    // Application specific
    xIN_PickPiece : BOOL; (* signal from the pick and place element
                             the number of picked signal depend on the recipe *)
    xIN_RotTableBlockedByPnp : BOOL; // Is the pick and place blocking the rotary table?
END_VAR
VAR_OUTPUT
    (* standart Ausgänge *)
    xOUT_ErrFlag  : BOOL;           // Error Flag 
    xOUT_Busy     : BOOL;           // Baustein befindet sich im Ablauf 
    xOUT_Done     : BOOL;           // Baustein hat den Ablauf beendet 		
    xOUT_Ready    : BOOL;           // Ready to begin, should be the same state as done	
    xOUT_Timeout  : BOOL;           // Timeout FB 
    xOUT_InitDone : BOOL;           // initialisierung fertig
    xOUT_Wait     : BOOL;           // Wartet auf Bedingung
    iOUT_Step     : ST125_Feeder_e; // Aktueller Schritt 
    sOUT_Step     : STRING;         // Aktueller Schritt but in string format
    bOUT_Error    : BYTE;           // Fehlernummer

    // Application specific
    xOUT_PceReadyToPick : BOOL; // the piece(s) is/are ready to picked
END_VAR
VAR
    (* Standard *)
    (* Schritt *)
    iLastStep : ST125_Feeder_e; // Merker letzter Schritt 
    iPreStep  : ST125_Feeder_e; // Schritt zurück nach Alarm 
    iAktStep  : ST125_Feeder_e; // aktueller Schritt

    // Trigger Starten 
    rtSTART : R_TRIG;
    // Timer TimeOut 
    TON_Timeout : TON;

    (* Bausteine *)

    // Application specific
    fb_axis125_10W               : FB_AxisLMturn_V1_1;
    simu_axis125_10W             : FB_Simu_AxisLM_V1_1;
    fb_feeder                    : FB_Feeder2Sensors;
    fifo                         : FB_Fifo(3);
    simu_feeder                  : FB_Simu_Feeder; // simulation of a feeder
    simu_fifo_feeder_to_rotTable : FB_Fifo(30);    // fifo to hold a piece
    rtPutPiece                   : R_TRIG;         // trigger to add a piece

    rtPick : R_TRIG; // r_trig signal from the pick and place machine

    iCurrentTableIndex : INT; // current table index
    iSearchIndex       : INT; (* Initialization index TO see how many element we have AT startup
                                 or after an alarm *)

    xPieceInSeparator      : BOOL; // The piece is at the entry of the round table
    xPieceWrongInSeparator : BOOL; // A piece is detected at the separator but it is the wrong one

    // This ton is used to ensure that the piece is completely inside
    // the entry of the round table so we are sure that we mesure correctly the piece up to
    // the top
    TON_waitForControl : TON;

END_VAR
VAR CONSTANT
    MAX_SEARCH_TURN : INT := 3; // maximum search number

    FEEDER_SIMULATION : BOOL := FALSE; // Simulate this code
END_VAR

(*******************************************************************)
(* Trigger  *)
(*******************************************************************)
(* Zurücksetzen *)
IF xIN_RESET THEN
    iPreStep  := ST125_Feeder_e.RESET;
    iOUT_Step := ST125_Feeder_e.RESET;
END_IF;

(* Error Quittieren *)
IF (bOUT_Error <> 0) AND xIN_Quit THEN
    xOUT_ErrFlag := FALSE;
    bOUT_Error   := 0;
    iOUT_Step    := iPreStep;
END_IF;

iCurrentTableIndex := iCurrentTableIndex MOD 3;

(*******************************************************************)
(* Timer *)
(*******************************************************************)
TON_Timeout(IN := xIN_NextStep AND (iLastStep = iOUT_Step) (*todo FG *) ,
            PT := tIN_Timeout);

xPieceInSeparator := (IN.AI21_ST125_piece_height < _20_AUTO.recipe.st125.diPieceGoodMaxHeight) AND
                     (IN.AI21_ST125_piece_height > _20_AUTO.recipe.st125.diPieceGoodMinHeight);

xPieceWrongInSeparator := (IN.AI21_ST125_piece_height < _20_AUTO.recipe.st125.diPieceWrongMaxHeight) AND
                          (IN.AI21_ST125_piece_height > _20_AUTO.recipe.st125.diPieceWrongMinHeight);

TON_waitForControl(IN := xPieceInSeparator,
                   PT := DINT_TO_TIME(_20_AUTO.recipe.st125.TON_WaitPieceTime));

(*******************************************************************)
(* Bausteine *)
(*******************************************************************)

fb_feeder(xIN_Enable                := enIN_State = enState.StateAUTO OR enIN_State = enState.StateSTEP,
          xIN_PieceInEnd            := IO_BOX.I8401_ST125_maximum_wf,
          xIN_PieceMax              := IO_BOX.I8401_ST125_maximum_wf,
          xIN_InSimulation          := FEEDER_SIMULATION AND CONST.USE_SIMULATION,
          refIN_SimulatedFifo       := simu_fifo_feeder_to_rotTable,
          iIN_FifoSetMaxSensorValue := 20,
          diIN_SignlFilter_ms       := _20_AUTO.recipe.st125.FeederConfig.InFilterDelay,
          diIN_StartDelay_ms        := _20_AUTO.recipe.st125.FeederConfig.StartDelay,
          diIN_StopDelay_ms         := _20_AUTO.recipe.st125.FeederConfig.StopDelay,
          diIN_EmptyDelay_ms        := _20_AUTO.recipe.st125.FeederConfig.EmptyDelay);

simu_feeder(xIN_Enable         := fb_feeder.xOUT_EnableFeeder AND FEEDER_SIMULATION AND CONST.USE_SIMULATION,
            xIN_PceSensor      := fb_feeder.xIN_PieceMax,
            tIN_NewPieceTime   := 500,
            iIN_WaitTimeMin_ms := 500,
            iIN_WaitTimeMax_ms := 1000);

rtPick(CLK := xIN_PickPiece);
rtPutPiece(CLK := simu_feeder.xOUT_NewPiece);

IF rtPutPiece.Q AND NOT simu_fifo_feeder_to_rotTable.IsFull() THEN
    simu_fifo_feeder_to_rotTable.Put(1);
END_IF

IF ST125_Feeder_e.Init_simu_home_table = iOUT_Step THEN
    fb_axis125_10W.rIN_Position := TO_REAL(120.0 - LMOD(ST125_Axis.axis125_10W.rActPos, 120.0));

ELSE
    fb_axis125_10W.rIN_Position := 120.0;

END_IF

simu_axis125_10W(xIN_Enable          := FEEDER_SIMULATION AND CONST.USE_SIMULATION,
                 wIN_AxisState       := ST125_Axis.axis125_10W.wState,
                 bIN_AxisCntr        := fb_axis125_10W.bOUT_AxisCntr,
                 udiIN_HomingTime_ms := 1000,
                 pIN_axisSimu        := ADR(SIMU.axis_ref[Axis_e.ST125_10W]),
                 pIN_axisHW          := ADR(ST125_Axis.axis125_10W.axis),
                 rIN_PosActual       := fb_axis125_10W.rOUT_ActPos,
                 rIN_PosMax          := ST125_Axis.const125_10W.POS_MAX,
                 rIN_PosMin          := ST125_Axis.const125_10W.POS_MIN,
                 rIN_PixMax          := 0,
                 rIN_PixMin          := 0);

fb_axis125_10W(enIN_State     := enIN_State,
               parIN_Buttons  := ADR(AXIS.btTeachArAxis[Axis_e.ST125_10W]),
               xIN_DisButtons :=,
               xIN_Quit       := xIN_Quit,
               xIN_PARAMok    := TRUE,
               xIN_FREE       := NOT xIN_RotTableBlockedByPnp,
               xIN_FREE_HOME  := TRUE,
               rIN_POSMIN     := ST125_Axis.const125_10W.POS_MIN,
               rIN_POSMAX     := ST125_Axis.const125_10W.POS_MAX,
               rIN_VELOMAX    := ST125_Axis.const125_10W.VELO_MAX,
               rIN_VELOMANU   := ST125_Axis.const125_10W.VELO_MANU,
               rIN_VELOOPEN   := ST125_Axis.const125_10W.VELO_MANU / 4,
               rIN_JogInc     := AXIS.rTeachIncAxis,
               xIN_Execute    := ST125_Feeder_e.Init_set_table_pos = iOUT_Step OR
                                 ST125_Feeder_e.Init_table_go_to_zero = iOUT_Step OR
                                 ST125_Feeder_e.Init_simu_home_table = iOUT_Step OR
                                 ST125_Feeder_e.load_piece = iOUT_Step OR
                                 ST125_Feeder_e.wait_rotary_table_done = iOUT_Step,
               xIN_Relative     := fb_axis125_10W.xIN_Execute,
               xIN_STOP         := FALSE,
               xIN_OFF          := FALSE,
               rIN_Position     :=, // Is set above
               rIN_Velocity     := TO_REAL(100.0),
               rIN_Acceleration := TO_REAL(2160.0),
               rIN_Deceleration := TO_REAL(2160.0),
               rIN_Jerk         := TO_REAL(720000.0),
               xIN_Home         := ST125_feeder_e.Init_home_table = iOUT_Step,
               xIN_Reset        := xIN_Reset OR ST125_feeder_e.RESET = iOUT_Step,
               // The simu fb gives us the hardware signal when we are not in simulation
               wAxisState    := simu_axis125_10W.wOUT_AxisState,
               bOUT_AxisCntr => ST125_Axis.axis125_10W.bCtrlHi,
               rOUT_ActPos   =>, // leave empty, rActPos must be set using the modulo
               axisIN_REF    := simu_axis125_10W.pOUT_axisRef^);

ST125_Axis.axis125_10W.rActPos := LREAL_TO_REAL(simu_axis125_10W.pOUT_axisRef^.NcToPlc.ModuloActPos);

(*******************************************************************)
(* OUTPUTS *)
(*******************************************************************)
// Error Flag 
xOUT_ErrFlag := (bOUT_Error <> 0) OR (ST125_Feeder_e.ERROR = iOUT_Step);
// Baustein befindet sich im Ablauf 
xOUT_Busy := (iOUT_Step > ST125_Feeder_e.READY) AND (iOUT_Step < ST125_Feeder_e.DONE);
// Baustein hat den Ablauf beendet
xOUT_Done := (iOUT_Step = ST125_Feeder_e.DONE);
// Process ready
xOUT_Ready := (iOUT_Step = ST125_Feeder_e.READY);
// Timeout FB 				 		
xOUT_Timeout := TON_Timeout.Q;
// Itialisierung fertig			
xOUT_InitDone := (iOUT_Step = ST125_Feeder_e.READY);
// Aktueller Schritt			
iOUT_Step := iOUT_Step; //Im Ablauf gesetzt		
sOUT_Step := TO_STRING(iOUT_Step);
//Fehlernummer	 
bOUT_Error := bOUT_Error; //Im Ablauf/FB gesetzt	
(* Warte (alle Schritte wo auf FG oder Teile gewartet wird) *)
xOUT_Wait := (iOUT_Step = ST125_Feeder_e.DONE) OR
             (iOUT_Step = ST125_Feeder_e.READY);

IO_BOX.Q8402_ST125_freigabe_wf := fb_feeder.xOUT_EnableFeeder AND NOT (FEEDER_SIMULATION AND CONST.USE_SIMULATION);

IO_BOX.Q8400_ST125_freigabe_REO :=
    (IO_BOX.Q8402_ST125_freigabe_wf OR
    (ST125_Feeder_e.wait_on_a_piece = iOUT_Step) OR
    (ST125_Feeder_e.DONE = iOUT_Step AND NOT xPieceInSeparator)) AND
    NOT (FEEDER_SIMULATION AND CONST.USE_SIMULATION);

(*******************************************************************)
(* Ablauf *)
(*******************************************************************)

(* Sperren *)
IF xIN_Sperre THEN
    iPreStep  := ST125_Feeder_e.RESET;
    iOUT_Step := ST125_Feeder_e.RESET;
    RETURN;
END_IF;

(* Schritt Merker *)
IF iAktStep <> iOUT_Step THEN
    iLastStep := iAktStep;
    iAktStep  := iOUT_Step;
END_IF

(* START *)
rtSTART(CLK := xIN_Start);

IF 0 = bOUT_Error THEN
    IF fb_axis125_10W.xOUT_ErrFlag THEN 
        bOUT_Error := ST125_Alarm_e.Axis_120_10W_error;
        iPreStep   := ST145_Feeder_e.INIT;
		
    ELSIF fb_feeder.xOUT_Empty THEN
        bOUT_Error := ST125_Alarm_e.Feeder_empty;
        iPreStep   := ST145_Feeder_e.READY;
		
	ELSIF IN.I504_distanzsensor_verschmutzung_125 THEN
        bOUT_Error := ST125_Alarm_e.Distance_sensor_dirty;
        iPreStep   := ST145_Feeder_e.INIT;
	
    END_IF
ELSIF iOUT_Step < ST125_Feeder_e.ERROR THEN
    iOUT_Step := ST125_Feeder_e.ERROR;
END_IF

(*******************************************************************)
(* Schrittkette  *)
(*******************************************************************)
CASE iOUT_Step OF

(***** RESET *****)
ST125_Feeder_e.RESET: (* Schritt 0-99 *)
    //Initialisierungen
    //Start Init Ablauf
    IF xIN_Init THEN
        iOUT_Step := ST125_Feeder_e.INIT;
        //Start Manu Ablauf
    ELSIF enIN_State = StateMANU AND xIN_NextStep THEN
        iOUT_Step := ST125_Feeder_e.INIT;
    END_IF;

(***** INIT *****)
ST125_Feeder_e.INIT: (* Grundstellung ? *)
    IF NOT xIN_RotTableBlockedByPnp THEN
        iOUT_Step := ST125_Feeder_e.Init_home_table;
    END_IF

ST125_Feeder_e.Init_home_table:
    IF fb_axis125_10W.xOUT_HOMED THEN
        iCurrentTableIndex := 0;

        IF FEEDER_SIMULATION AND CONST.USE_SIMULATION THEN
            iOUT_Step := ST125_Feeder_e.Init_simu_home_table;
        ELSE
            iOUT_Step := ST125_Feeder_e.Init_reset_search_index;
        END_IF
    END_IF

ST125_Feeder_e.Init_simu_home_table:
    IF fb_axis125_10W.xOUT_DONE THEN
        iOUT_Step := ST125_Feeder_e.Init_reset_search_index;
    END_IF

// unused, done by the drive itself, see drive configuration
ST125_Feeder_e.Init_table_go_to_zero:
    IF fb_axis125_10W.xOUT_DONE THEN
        iOUT_Step := ST125_Feeder_e.Init_reset_search_index;
    END_IF

ST125_Feeder_e.Init_reset_search_index:
    iSearchIndex := 0;
    fifo.Empty();
    iOUT_Step := ST125_Feeder_e.READY; // Bypass search algorithm, unusful

ST125_Feeder_e.Init_set_table_pos:
    IF fb_axis125_10W.xOUT_DONE THEN
        iCurrentTableIndex := iCurrentTableIndex + 1;
        iOUT_Step          := ST125_Feeder_e.Init_see_if_piece_there;
    END_IF

ST125_Feeder_e.Init_see_if_piece_there:
    IF simu_feeder.xOUT_NewPiece THEN
        fifo.Put(1);
    END_IF

    IF iSearchIndex < MAX_SEARCH_TURN THEN
        iOUT_Step    := ST125_Feeder_e.Init_set_table_pos;
        iSearchIndex := iSearchIndex + 1;
    ELSE
        iOUT_Step := ST125_Feeder_e.READY;
    END_IF

(***** READY / INIT DONE *****)
ST125_Feeder_e.READY: (* Start AUTO,END,LEER,STEP *)
    IF xIN_Start THEN //IF rtSTART.Q THEN
        iOUT_Step := ST125_Feeder_e.START;
    END_IF

(***** START  ZYKLISCH *****)
ST125_Feeder_e.START: (*  *)
    IF xIN_NextStep AND pxFG_Freigabe^ THEN
        iOUT_Step := ST125_Feeder_e.check_if_feeding_necessary;
    END_IF;

ST125_Feeder_e.check_if_feeding_necessary:
    IF fifo.IsFull() THEN
        iOUT_Step := ST125_Feeder_e.DONE;
    ELSE
        iOUT_Step := ST125_Feeder_e.wait_on_a_piece;
    END_IF

ST125_Feeder_e.wait_on_a_piece:
    IF (FEEDER_SIMULATION AND CONST.USE_SIMULATION AND NOT simu_fifo_feeder_to_rotTable.IsEmpty()) OR
       (NOT (FEEDER_SIMULATION AND CONST.USE_SIMULATION) AND TON_waitForControl.Q) THEN
        iOUT_Step := ST125_Feeder_e.load_piece;
        simu_fifo_feeder_to_rotTable.Pop(1);
    END_IF

ST125_Feeder_e.load_piece:
    IF NOT fb_axis125_10W.xOUT_DONE THEN
        iOUT_Step := ST125_Feeder_e.wait_rotary_table_done;
    END_IF

ST125_Feeder_e.wait_rotary_table_done:
    IF fb_axis125_10W.xOUT_DONE THEN
        fifo.Put(1);
        iOUT_Step := ST125_Feeder_e.check_if_feeding_necessary;
    END_IF

(***** DONE *****)
ST125_Feeder_e.DONE: (* Letzter Schritt  *)
    IF rtPick.Q THEN
        fifo.Pop(TO_INT(_20_AUTO.recipe.st125.xUseVerLeft));
        fifo.Pop(TO_INT(_20_AUTO.recipe.st125.xUseVerRight));
    END_IF

    IF NOT xIN_AlarmAktiv THEN
        //AUTO
        IF (enIN_State = StateAUTO) AND xIN_RestartCYCL AND NOT fifo.IsFull() THEN
            iOUT_Step := ST125_Feeder_e.START;
            //STEP / END / LEERFAHREN restart
        ELSIF (enIN_State < StateAUTO) AND (enIN_State >= enState.StateSTEP) AND xIN_RestartCYCL AND NOT fifo.IsFull()
            THEN
            iOUT_Step := ST125_Feeder_e.START;
            //STEP / END / LEERFAHREN fertig
        ELSIF (enIN_State = StateREADY) THEN
            iOUT_Step := ST125_Feeder_e.READY;
        END_IF;
    END_IF;

(************ ERROR *************)
ST125_Feeder_e.ERROR: (* ERROR *) ;

END_CASE;

END_FUNCTION_BLOCK

// ---- POUs/20_AUTO/ST125/POU_ALARM_125.TcPOU
PROGRAM POU_ALARM_125
VAR_INPUT
    xIN_QUIT      : BOOL; // Alarm quittieren
    iIN_ArraySize : INT;
    pstrIN_ALARM  : POINTER TO structAlarm;       // Array Alarmstruktur
    refPOU        : REFERENCE TO FB_AUT_ABSTRACT; // the POU to test
END_VAR
VAR_OUTPUT
    xOUT_AL_ST : BOOL; // Alarm Station aktiv
END_VAR
VAR
    //Alarmbaustein
    _FB_ALARM_ST : FB_ALARM;
    //Local
    iIndex : INT; // Index For Schleife	
END_VAR
VAR CONSTANT
    sDefString : STRING := 'Error ST120,'; // Station #
END_VAR

(********************** INITIALISIERE VARIABLEN ****************************)
FOR iIndex := 0 TO iIN_ArraySize - 1 DO
    pstrIN_ALARM[iIndex].xAlarmIN   := FALSE;
    pstrIN_ALARM[iIndex].xAlarmOFF  := FALSE;
    pstrIN_ALARM[iIndex].xAlarmSAVE := TRUE;
    pstrIN_ALARM[iIndex].xAlarmQUIT := xIN_QUIT;
    pstrIN_ALARM[iIndex].tAlarmVERZ := T#100MS;
    pstrIN_ALARM[iIndex].sAlarmText := '';
    pstrIN_ALARM[iIndex].bAlarmNr   := 0;
END_FOR

(********************** ALARME ****************************)
pstrIN_ALARM[0].xAlarmIN   := (refPOU.bOUT_ErrorNum = ST120_Alarm_e.Axis_120_01Y_error);
pstrIN_ALARM[0].sAlarmText := CONCAT(sDefString, ' Axis 01Y in error');
pstrIN_ALARM[0].bAlarmNr   := 0;

pstrIN_ALARM[1].xAlarmIN   := (refPOU.bOUT_ErrorNum = ST120_Alarm_e.Axis_120_02Z_error);
pstrIN_ALARM[1].sAlarmText := CONCAT(sDefString, ' Axis 02Z in error');
pstrIN_ALARM[1].bAlarmNr   := 0;

pstrIN_ALARM[2].xAlarmIN   := (refPOU.bOUT_ErrorNum = ST120_Alarm_e.Cylinder_griper_left);
pstrIN_ALARM[2].sAlarmText := CONCAT(sDefString, ' Cylinder .05 gripper right');
pstrIN_ALARM[2].bAlarmNr   := 0;

pstrIN_ALARM[3].xAlarmIN   := (refPOU.bOUT_ErrorNum = ST120_Alarm_e.Cylinder_griper_right);
pstrIN_ALARM[3].sAlarmText := CONCAT(sDefString, ' Cylinder .06 gripper left');
pstrIN_ALARM[3].bAlarmNr   := 0;

pstrIN_ALARM[7].xAlarmIN   := (refPOU.bOUT_ErrorNum = ST120_Alarm_e.Feeder_error);
pstrIN_ALARM[7].sAlarmText := CONCAT(sDefString, ' One part of the feeder is in error');
pstrIN_ALARM[7].bAlarmNr   := 0;

pstrIN_ALARM[8].xAlarmIN   := (refPOU.bOUT_ErrorNum = ST120_Alarm_e.Piece_in_unused_griper);
pstrIN_ALARM[8].sAlarmText := CONCAT(sDefString, ' One part is handled by a unused griper');
pstrIN_ALARM[8].bAlarmNr   := 0;

pstrIN_ALARM[9].xAlarmIN   := (refPOU.bOUT_ErrorNum = ST120_Alarm_e.Piece_missing_left_griper);
pstrIN_ALARM[9].sAlarmText := CONCAT(sDefString, ' A piece is missing in the left griper');
pstrIN_ALARM[9].bAlarmNr   := 0;

pstrIN_ALARM[10].xAlarmIN   := (refPOU.bOUT_ErrorNum = ST120_Alarm_e.Piece_missing_right_griper);
pstrIN_ALARM[10].sAlarmText := CONCAT(sDefString, ' A piece is missing in the right griper');
pstrIN_ALARM[10].bAlarmNr   := 0;

pstrIN_ALARM[11].xAlarmIN   := (refPOU.bOUT_ErrorNum = ST120_Alarm_e.Feeder_empty);
pstrIN_ALARM[11].sAlarmText := CONCAT(sDefString, ' The feeder is empty');
pstrIN_ALARM[11].bAlarmNr   := 0;

(********************** ALARM FB ****************************)
_FB_ALARM_ST(pstrIN_Alarm  := pstrIN_ALARM,
             iIN_ArraySize := ST120_Alarm_e._max);

(********************** ALARM FB ****************************)
xOUT_AL_ST := FALSE;

FOR iIndex := 0 TO iIN_ArraySize - 1 DO
    IF pstrIN_ALARM[iIndex].xAlarmOUT THEN
        xOUT_AL_ST := TRUE;
    END_IF
END_FOR

END_PROGRAM

// ---- POUs/20_AUTO/ST128/FB_AUT_128.TcPOU
FUNCTION_BLOCK FB_AUT_128 EXTENDS FB_AUT_ABSTRACT
(****************************************************************************)
(*	POU_AUT_zxx			Bausteinaufrufe Station	zxx							*)
(*	Status				ungetestet											*)
(*  Version:			1.0													*)
(*	Beschrieb:																*)
(*																			*)
(*	Abläufe:			FB_ABLzxxA		Hauptablauf							*)
(*																			*)
(*																			*)
(* 	25.09.2019/Dj															*)
(****************************************************************************)
(*	dd.mm.yyyy   KZ    x.y			Beschrieb								*)
(****************************************************************************)
VAR_INPUT
    (* spezifische Eingänge *)

END_VAR
VAR_OUTPUT
    (* spezifische Ausgänge *)

END_VAR
VAR
    (* Bausteine *)
    fb_TubeCapCheck : FB_ABL_128_TubeCapCheck; // 
END_VAR

(*******************************************************************)
(* Timer *)
(*******************************************************************)

(*******************************************************************)
(* Flanken / Merker *)
(*******************************************************************)
//MANU CYCLE
IF (enIN_State = StateMANU) AND xIN_ManuCycle THEN
    xManuCycle := TRUE;
END_IF;

IF (enIN_State <> StateMANU) OR xOUT_Done THEN
    xManuCycle := FALSE;
END_IF

//NEXT STEP
xNextStep := (enIN_State > StateSTEP) OR
             ((enIN_State = StateSTEP) AND xIN_Step) OR
             ((enIN_State = StateMANU) AND xManuCycle);

//RESET
xReset := (enIN_State < StateREADY) AND (enIN_State <> StateINIT) AND NOT xManuCycle;

(*******************************************************************)
(* Bausteinaufrufe Abläufe *)
(*******************************************************************)

xRelease := MAIN.MoverMan.IsProcessUsed(THIS^);

fb_TubeCapCheck(xIN_Reset       := xReset,
                xIN_Init        := xIN_Init,
                xIN_Quit        := xIN_Quit,
                xIN_Start       := enIN_State >= enState.StateLEER AND xRelease,
                xIN_Sperre      := NOT xIN_On,
                xIN_NextStep    := xNextStep,
                xIN_AlarmAktiv  := xIN_AlarmAktiv,
                xIN_DryCycle    := xIN_DryCycle,
                xIN_RestartCYCL := enIN_State >= enState.StateLEER,
                enIN_State      := enIN_State,
                tIN_Timeout     := tIN_Timeout,
                pxFG_Freigabe   := ADR(xRelease),
                Mover           := THIS^.Mover);

(*******************************************************************)
(* Mover reset flags *)
(*******************************************************************)

(*******************************************************************)
(* OUTPUT *)
(*******************************************************************)
xOUT_InitDone := fb_TubeCapCheck.xOUT_InitDone;
xOUT_Ready    := fb_TubeCapCheck.xOUT_Ready;
xOUT_Done     := fb_TubeCapCheck.xOUT_Done;
xOUT_ErrFlag  := fb_TubeCapCheck.xOUT_ErrFlag;
xOUT_Wait     := fb_TubeCapCheck.xOUT_Wait;
xOUT_AlarmST  := xOUT_ErrFlag;

(*******************************************************************)
(* Bausteinaufruf Error Station *)
(*******************************************************************)
// POU_ERR_VORLAGE(xIN_QUIT:=xIN_Quit , pstrArIN_ALARM:=ADR(HMI.strArALARM[1]));

(* % of completion of the process *)
PROPERTY iCompletionPC : INT
GET
iCompletionPC := THIS^.fb_TubeCapCheck.iOUT_ProcessCompletion;
END_GET
END_PROPERTY

PROPERTY ProcessExecution : ProcessExecution_e
GET
ProcessExecution := THIS^._ProcessExecution;
END_GET
SET
THIS^._ProcessExecution := ProcessExecution;
END_SET
END_PROPERTY

PROPERTY xBusy : BOOL
GET
xBusy := THIS^.fb_TubeCapCheck.xOUT_Busy;
END_GET
SET
END_SET
END_PROPERTY

PROPERTY xDone : BOOL
GET
xDone := THIS^.fb_TubeCapCheck.xOUT_Ready OR THIS^.fb_TubeCapCheck.xOUT_Done;
END_GET
END_PROPERTY

PROPERTY xMoverPathFree : BOOL
GET
xMoverPathFree := THIS^.fb_TubeCapCheck.xOUT_MoverFree OR THIS^.fb_TubeCapCheck.xOUT_Ready OR THIS^.fb_TubeCapCheck.xOUT_Done;
END_GET
END_PROPERTY

PROPERTY xMoverShouldLeave : BOOL
GET
xMoverShouldLeave := THIS^.fb_TubeCapCheck.iOUT_Step = ST128_TubeCapCheck_e.SYNC_MOVER_LEAVE;
END_GET
END_PROPERTY

END_FUNCTION_BLOCK

// ---- POUs/20_AUTO/ST128/FB_ABL_128_TubeCapCheck.TcPOU
FUNCTION_BLOCK FB_ABL_128_TubeCapCheck
(****************************************************************************************)
(*	TITEL				laden kristall- Modul	    										*)
(*	Status				ungetestet                         								*)
(*	Beschrieb:			Ablaufbeschreibung												*)
(*																						*)
(*	Steps:	self-explained using enum													*)
(***********************************Revisionen*******************************************)
(*	see github blames																	*)
(****************************************************************************************)

VAR_INPUT
    xIN_Reset       : BOOL;          // Schrittkette zurücksetzen 
    xIN_Init        : BOOL;          // Initialisieren
    xIN_Quit        : BOOL;          // Fehler quittieren 
    xIN_Start       : BOOL;          // Startbefehl
    xIN_Sperre      : BOOL;          // FB Sperren 
    xIN_NextStep    : BOOL;          // Nächsten Schritt ausführen 
    xIN_AlarmAktiv  : BOOL;          // Anlage hat Alarm
    xIN_DryCycle    : BOOL;          // Fahren ohne Teile
    xIN_RestartCYCL : BOOL;          // Zyklus erneut starten im STEP: END: LEERFAHREN
    enIN_State      : enState;       // Status Anlage
    tIN_Timeout     : TIME := T#10s; // Timout

    pxFG_Freigabe : POINTER TO BOOL; //Freigabe von Station

    // Application specific
    Mover : REFERENCE TO FB_Mover;
END_VAR
VAR_OUTPUT
    (* standart Ausgänge *)
    xOUT_ErrFlag  : BOOL;                 // Error Flag 
    xOUT_Busy     : BOOL;                 // Baustein befindet sich im Ablauf 
    xOUT_Done     : BOOL;                 // Baustein hat den Ablauf beendet 		
    xOUT_Ready    : BOOL;                 // Ready to begin: should be the same state as done	
    xOUT_Timeout  : BOOL;                 // Timeout FB 
    xOUT_InitDone : BOOL;                 // initialisierung fertig
    xOUT_Wait     : BOOL;                 // Wartet auf Bedingung
    iOUT_Step     : ST128_TubeCapCheck_e; // Aktueller Schritt 
    sOUT_Step     : STRING;               // Aktueller Schritt but in string format
    bOUT_Error    : BYTE;                 // Fehlernummer

    iOUT_ProcessCompletion : INT;  //process completion: express in % (0-100)
    xOUT_MoverFree         : BOOL; // The mover is free to move

END_VAR
VAR
    (* Standard *)
    (* Schritt *)
    iLastStep : ST128_TubeCapCheck_e; // Merker letzter Schritt 
    iPreStep  : ST128_TubeCapCheck_e; // Schritt zurück nach Alarm 
    iAktStep  : ST128_TubeCapCheck_e; // aktueller Schritt

    // Trigger Starten 
    rtSTART : R_TRIG;
    // Timer TimeOut 
    TON_Timeout : TON;

    (* Bausteine *)
    ton_WaitInPosMin : TON;  // protect the inpos flag to come to early
    capFoundRight    : BOOL; // TRUE when all measured level are OK
    capFoundLeft     : BOOL; // TRUE when all measured level are OK

    visu_shuttle_x_position : LREAL; // position of the shuttle used in visu

END_VAR
VAR CONSTANT
    TUBE_CAP_CHECK_SIMULATION : BOOL := FALSE; // Set to TRUE to simulate this part of the program
END_VAR

(*******************************************************************)
(* Trigger  *)
(*******************************************************************)
(* Zurücksetzen *)
IF xIN_RESET THEN
    iPreStep  := ST128_TubeCapCheck_e.RESET;
    iOUT_Step := ST128_TubeCapCheck_e.RESET;
END_IF;

(* Error Quittieren *)
IF (bOUT_Error <> 0) AND xIN_Quit THEN
    xOUT_ErrFlag := FALSE;
    bOUT_Error   := 0;
    iOUT_Step    := iPreStep; // iPreStep;
END_IF;

(*******************************************************************)
(* Timer *)
(*******************************************************************)
TON_Timeout(IN := xIN_NextStep AND (iLastStep = iOUT_Step) (*todo FG *) ,
            PT := tIN_Timeout);

ton_WaitInPosMin(IN := __ISVALIDREF(Mover) AND_THEN Mover.IsInStationPos(), PT := T#100MS);

(*******************************************************************)
(* Bausteine *)
(*******************************************************************)
IF (iOUT_Step = ST128_TubeCapCheck_e.Wait_move_and_check_tube_cap_right OR
   iOUT_Step = ST128_TubeCapCheck_e.Move_shuttle_relative_right) AND
   IO_BOX.I2000_ST128_filterhut_vorhanden THEN
    capFoundRight := TRUE;
END_IF

IF (iOUT_Step = ST128_TubeCapCheck_e.Wait_move_and_check_tube_cap_left OR
   iOUT_Step = ST128_TubeCapCheck_e.Move_shuttle_relative_left) AND
   IO_BOX.I2000_ST128_filterhut_vorhanden THEN
    capFoundLeft := TRUE;
END_IF

(*******************************************************************)
(* OUTPUTS *)
(*******************************************************************)
// Error Flag 
xOUT_ErrFlag := (bOUT_Error <> 0) OR (ST128_TubeCapCheck_e.ERROR = iOUT_Step);
// Baustein befindet sich im Ablauf 
xOUT_Busy := (iOUT_Step > ST128_TubeCapCheck_e.READY) AND (iOUT_Step < ST128_TubeCapCheck_e.DONE);
// Baustein hat den Ablauf beendet
xOUT_Done := (iOUT_Step = ST128_TubeCapCheck_e.DONE);
// Process ready
xOUT_Ready := (iOUT_Step = ST128_TubeCapCheck_e.READY);
// Timeout FB 				 		
xOUT_Timeout := TON_Timeout.Q;
// Itialisierung fertig			
xOUT_InitDone := (iOUT_Step = ST128_TubeCapCheck_e.READY) OR
                 (iOUT_Step = ST128_TubeCapCheck_e.DONE);

// Aktueller Schritt			
iOUT_Step := iOUT_Step; //Im Ablauf gesetzt		
sOUT_Step := TO_STRING(iOUT_Step);
//Fehlernummer	 
bOUT_Error := bOUT_Error; //Im Ablauf/FB gesetzt	
(* Warte (alle Schritte wo auf FG oder Teile gewartet wird) *)
xOUT_Wait := (iOUT_Step = ST128_TubeCapCheck_e.DONE) OR
             (iOUT_Step = ST128_TubeCapCheck_e.READY) OR
             (iOUT_Step = ST128_TubeCapCheck_e.START) OR
             (iOUT_Step = ST128_TubeCapCheck_e.waitOnMover) OR
             (iOUT_Step = ST128_TubeCapCheck_e.SYNC_MOVER_LEAVE);

xOUT_MoverFree :=
    NOT ((iOUT_Step >= ST128_TubeCapCheck_e.MOVER_NEEDED_OP) AND (iOUT_Step < ST128_TubeCapCheck_e.MOVER_FREE_OP)) AND
    (iOUT_Step >= ST128_TubeCapCheck_e.READY) AND
    (iOUT_Step < ST128_TubeCapCheck_e.ERROR);

iOUT_ProcessCompletion := F_GetPercent_2(iOUT_Step,
                                         ST128_TubeCapCheck_e.waitOnMover,
                                         ST128_TubeCapCheck_e.DONE,
                                         ST128_TubeCapCheck_e.waitOnMover,
                                         ST128_TubeCapCheck_e.DONE);

(*******************************************************************)
(* Ablauf *)
(*******************************************************************)

(* Sperren *)
IF xIN_Sperre THEN
    iPreStep  := ST128_TubeCapCheck_e.RESET;
    iOUT_Step := ST128_TubeCapCheck_e.RESET;
    RETURN;
END_IF;

(* Schritt Merker *)
IF iAktStep <> iOUT_Step THEN
    iLastStep := iAktStep;
    iAktStep  := iOUT_Step;
END_IF

(* START *)
rtSTART(CLK := xIN_Start);

IF __ISVALIDREF(Mover) THEN
    visu_shuttle_x_position := Mover.MovingProcessOffset;
ELSE
    visu_shuttle_x_position := 0.0;
END_IF

IF 0 = bOUT_Error THEN
    // put error conditions here
ELSIF iOUT_Step < ST128_TubeCapCheck_e.ERROR THEN
    iOUT_Step := ST128_TubeCapCheck_e.ERROR;
END_IF

(*******************************************************************)
(* Schrittkette  *)
(*******************************************************************)
CASE iOUT_Step OF

(***** RESET *****)
ST128_TubeCapCheck_e.RESET: (* Schritt 0-99 *)
    //Initialisierungen
    //Start Init Ablauf
    IF xIN_Init THEN
        iOUT_Step := ST128_TubeCapCheck_e.INIT;
        //Start Manu Ablauf
    ELSIF enIN_State = StateMANU AND xIN_NextStep THEN
        iOUT_Step := ST128_TubeCapCheck_e.INIT;
    END_IF;

(***** INIT *****)
ST128_TubeCapCheck_e.INIT: (* Grundstellung ? *)
    iOUT_Step := ST128_TubeCapCheck_e.READY;

(***** READY / INIT DONE *****)
ST128_TubeCapCheck_e.READY: (* Start AUTO:END:LEER:STEP *)
    IF xIN_Start THEN       //IF rtSTART.Q THEN
        iOUT_Step := ST128_TubeCapCheck_e.START;
    END_IF

(***** START  ZYKLISCH *****)
ST128_TubeCapCheck_e.START: (*  *)
    IF xIN_NextStep AND pxFG_Freigabe^ THEN
        iOUT_Step     := ST128_TubeCapCheck_e.waitOnMover;
        capFoundRight := FALSE;
        capFoundLeft  := FALSE;
    END_IF;

ST128_TubeCapCheck_e.waitOnMover:
    IF xIN_NextStep AND __ISVALIDREF(Mover) OR HMI.bArForceCyclusState[StationList_e.ST128] THEN
        IF Mover.GetLastStationDone() >= INT#128 THEN
            iOUT_Step := ST128_TubeCapCheck_e.SYNC_MOVER_LEAVE;
        ELSIF Mover.GetLastStationDone() < INT#125 THEN
            iOUT_Step := ST128_TubeCapCheck_e.SYNC_MOVER_LEAVE;
        ELSE
            iOUT_Step := ST128_TubeCapCheck_e.Move_shuttle_relative_right;
        END_IF
    END_IF

ST128_TubeCapCheck_e.Move_shuttle_relative_right:
    IF __ISVALIDREF(Mover) THEN
        IF Mover.MoveRelativeInsideStation(40.0) THEN
            iOUT_Step := ST128_TubeCapCheck_e.Wait_move_and_check_tube_cap_right;
            iPreStep  := ST128_TubeCapCheck_e.Wait_move_and_check_tube_cap_right;
        END_IF
    ELSE
        bOUT_Error := 10;
    END_IF

ST128_TubeCapCheck_e.Wait_move_and_check_tube_cap_right:
    IF xIN_NextStep AND __ISVALIDREF(Mover) AND_THEN ton_WaitInPosMin.Q THEN
        IF _20_AUTO.recipe.st128.xIsTypeMiniOrSmart THEN
            iOUT_Step := ST128_TubeCapCheck_e.Move_shuttle_to_pos_left;
        ELSE
            iOUT_Step := ST128_TubeCapCheck_e.Save_result_in_mover;
            iPreStep  := ST128_TubeCapCheck_e.Save_result_in_mover;
        END_IF
    END_IF

ST128_TubeCapCheck_e.Move_shuttle_to_pos_left:
    IF __ISVALIDREF(Mover) THEN
        IF Mover.MoveRelativeInsideStation(60.0) THEN
            iOUT_Step := ST128_TubeCapCheck_e.Wait_move_done_pos_left;
            iPreStep  := ST128_TubeCapCheck_e.Wait_move_done_pos_left;
        END_IF
    ELSE
        bOUT_Error := 11;
    END_IF

ST128_TubeCapCheck_e.Wait_move_done_pos_left:
    IF xIN_NextStep AND __ISVALIDREF(Mover) AND_THEN ton_WaitInPosMin.Q THEN
        iOUT_Step := ST128_TubeCapCheck_e.Move_shuttle_relative_left;
    END_IF

ST128_TubeCapCheck_e.Move_shuttle_relative_left:
    IF __ISVALIDREF(Mover) THEN
        IF Mover.MoveRelativeInsideStation(40.0) THEN
            iOUT_Step := ST128_TubeCapCheck_e.Wait_move_and_check_tube_cap_left;
            iPreStep  := ST128_TubeCapCheck_e.Wait_move_and_check_tube_cap_left;
        END_IF
    ELSE
        bOUT_Error := 12;
    END_IF

ST128_TubeCapCheck_e.Wait_move_and_check_tube_cap_left:
    IF xIN_NextStep AND __ISVALIDREF(Mover) AND_THEN ton_WaitInPosMin.Q THEN
        iOUT_Step := ST128_TubeCapCheck_e.Save_result_in_mover;
    END_IF

ST128_TubeCapCheck_e.Save_result_in_mover:
    IF (NOT capFoundRight OR
       (_20_AUTO.recipe.st128.xIsTypeMiniOrSmart AND NOT capFoundLeft)) AND
       NOT (TUBE_CAP_CHECK_SIMULATION AND CONST.USE_SIMULATION) THEN
        iOUT_Step := ST128_TubeCapCheck_e.ERROR;

        IF __ISVALIDREF(Mover) THEN

            IF NOT capFoundLeft AND NOT capFoundRight THEN
                Mover.SetErrorCode('128-B Left and Right');

            ELSIF capFoundLeft THEN
                Mover.SetErrorCode('128-B Left');

            ELSIF capFoundRight THEN
                Mover.SetErrorCode('128-B Right');

            ELSE
                ASSERT(0); // Read your code again, you should never go here !

            END_IF

            IF NOT Mover.SetLastStation(-128) THEN
                ASSERT(0);
            END_IF
        END_IF

        bOUT_Error := 1;
        iPreStep   := ST128_TubeCapCheck_e.SYNC_MOVER_LEAVE;
    ELSE
        iOUT_Step := ST128_TubeCapCheck_e.SYNC_MOVER_LEAVE;

        IF __ISVALIDREF(Mover) THEN
            IF NOT Mover.SetLastStation(128) THEN
                ASSERT(0);
            END_IF
        END_IF
    END_IF

ST128_TubeCapCheck_e.SYNC_MOVER_LEAVE:
    // The mover needs to be taken by MoverMan
    IF NOT __ISVALIDREF(Mover) THEN
        iOUT_Step := ST128_TubeCapCheck_e.DONE;
    END_IF

(***** DONE *****)
ST128_TubeCapCheck_e.DONE: (* Letzter Schritt  *)
    IF NOT xIN_AlarmAktiv THEN
        //AUTO
        IF (enIN_State = StateAUTO) AND xIN_RestartCYCL THEN
            iOUT_Step := ST128_TubeCapCheck_e.START;
            //STEP / END / LEERFAHREN restart
        ELSIF (enIN_State < StateAUTO) AND (enIN_State >= enState.StateSTEP) AND xIN_RestartCYCL THEN
            iOUT_Step := ST128_TubeCapCheck_e.START;
            //STEP / END / LEERFAHREN fertig
        ELSIF (enIN_State = StateREADY) THEN
            iOUT_Step := ST128_TubeCapCheck_e.READY;
        END_IF;
    END_IF;

(************ ERROR *************)
ST128_TubeCapCheck_e.ERROR: (* ERROR *) ;

END_CASE;

END_FUNCTION_BLOCK

// ---- POUs/20_AUTO/ST130/FB_AUT_130.TcPOU
FUNCTION_BLOCK FB_AUT_130 EXTENDS FB_AUT_ABSTRACT
(****************************************************************************)
(*	POU_AUT_zxx			Bausteinaufrufe Station	zxx							*)
(*	Status				ungetestet											*)
(*  Version:			1.0													*)
(*	Beschrieb:																*)
(*																			*)
(*	Abläufe:			FB_ABLzxxA		Hauptablauf							*)
(*																			*)
(*																			*)
(* 	25.09.2019/Dj															*)
(****************************************************************************)
(*	dd.mm.yyyy   KZ    x.y			Beschrieb								*)
(****************************************************************************)
VAR_INPUT
    (* spezifische Eingänge *)

END_VAR
VAR_OUTPUT
    (* spezifische Ausgänge *)

END_VAR
VAR
    (* Bausteine *)
    fb_Dose : FB_ABL_130_Dose;

    fb_stat : FB_AUT_Statistics;

END_VAR

(*******************************************************************)
(* Timer *)
(*******************************************************************)

(*******************************************************************)
(* Flanken / Merker *)
(*******************************************************************)
//MANU CYCLE
IF (enIN_State = StateMANU) AND xIN_ManuCycle THEN
    xManuCycle := TRUE;
END_IF;

IF (enIN_State <> StateMANU) OR xOUT_Done THEN
    xManuCycle := FALSE;
END_IF

//NEXT STEP
xNextStep := (enIN_State > StateSTEP) OR
             ((enIN_State = StateSTEP) AND xIN_Step) OR
             ((enIN_State = StateMANU) AND xManuCycle);

//RESET
xReset := (enIN_State < StateREADY) AND (enIN_State <> StateINIT) AND NOT xManuCycle;

(*******************************************************************)
(* Bausteinaufrufe Abläufe *)
(*******************************************************************)

xRelease := MAIN.MoverMan.IsProcessUsed(THIS^);

fb_Dose(xIN_Reset       := xReset,
        xIN_Init        := xIN_Init,
        xIN_Quit        := xIN_Quit,
        xIN_Start       := enIN_State >= enState.StateLEER AND xRelease,
        xIN_Sperre      := NOT xIN_On,
        xIN_NextStep    := xNextStep,
        xIN_AlarmAktiv  := xIN_AlarmAktiv,
        xIN_DryCycle    := xIN_DryCycle,
        xIN_RestartCYCL := enIN_State >= enState.StateLEER,
        enIN_State      := enIN_State,
        tIN_Timeout     := tIN_Timeout,
        pxFG_Freigabe   := ADR(xRelease),
        Mover           := THIS^.Mover);

fb_stat(xIN_Enable  := enState.StateAUTO = enIN_State,
        xIN_Waiting := fb_Dose.xOUT_Wait,
        xIN_Running := (fb_Dose.iOUT_Step >= ST130_Dose_e.START) AND
                       (fb_Dose.iOUT_Step <= ST130_Dose_e.DONE),
        // Since we use a mover system, a cycle is done when we are waiting on a mover
        xIN_Done := fb_Dose.iOUT_Step = ST130_Dose_e.waitOnMover);

(*******************************************************************)
(* Mover reset flags *)
(*******************************************************************)

(*******************************************************************)
(* OUTPUT *)
(*******************************************************************)
xOUT_InitDone := fb_Dose.xOUT_InitDone;
xOUT_Ready    := fb_Dose.xOUT_Ready;
xOUT_Done     := fb_Dose.xOUT_Done;
xOUT_ErrFlag  := fb_Dose.xOUT_ErrFlag;
xOUT_Wait     := fb_Dose.xOUT_Wait;
xOUT_AlarmST  := xOUT_ErrFlag;

(*******************************************************************)
(* Bausteinaufruf Error Station *)
(*******************************************************************)
// POU_ERR_VORLAGE(xIN_QUIT:=xIN_Quit , pstrArIN_ALARM:=ADR(HMI.strArALARM[1]));

(* % of completion of the process *)
PROPERTY iCompletionPC : INT
GET
iCompletionPC := THIS^.fb_Dose.iOUT_ProcessCompletion;
END_GET
END_PROPERTY

PROPERTY ProcessExecution : ProcessExecution_e
GET
ProcessExecution := THIS^._ProcessExecution;
END_GET
SET
THIS^._ProcessExecution := ProcessExecution;
END_SET
END_PROPERTY

PROPERTY xBusy : BOOL
GET
xBusy := THIS^.fb_Dose.xOUT_Busy;
END_GET
SET
END_SET
END_PROPERTY

PROPERTY xDone : BOOL
GET
xDone := THIS^.fb_Dose.xOUT_Ready OR THIS^.fb_Dose.xOUT_Done;
END_GET
END_PROPERTY

PROPERTY xMoverPathFree : BOOL
GET
xMoverPathFree := THIS^.fb_Dose.xOUT_MoverFree OR THIS^.fb_Dose.xOUT_Ready OR THIS^.fb_Dose.xOUT_Done;
END_GET
END_PROPERTY

PROPERTY xMoverShouldLeave : BOOL
GET
xMoverShouldLeave := THIS^.fb_Dose.iOUT_Step = ST130_Dose_e.SYNC_MOVER_LEAVE;
END_GET
END_PROPERTY

END_FUNCTION_BLOCK

// ---- POUs/20_AUTO/ST130/FB_ABL_130_Dose.TcPOU
FUNCTION_BLOCK FB_ABL_130_Dose
(****************************************************************************************)
(*	TITEL				laden kristall- Modul	    										*)
(*	Status				ungetestet                         								*)
(*	Beschrieb:			Ablaufbeschreibung												*)
(*																						*)
(*	Steps:	self-explained using enum													*)
(***********************************Revisionen*******************************************)
(*	see github blames																	*)
(****************************************************************************************)

VAR_INPUT
    xIN_Reset       : BOOL;          // Schrittkette zurücksetzen 
    xIN_Init        : BOOL;          // Initialisieren
    xIN_Quit        : BOOL;          // Fehler quittieren 
    xIN_Start       : BOOL;          // Startbefehl
    xIN_Sperre      : BOOL;          // FB Sperren 
    xIN_NextStep    : BOOL;          // Nächsten Schritt ausführen 
    xIN_AlarmAktiv  : BOOL;          // Anlage hat Alarm
    xIN_DryCycle    : BOOL;          // Fahren ohne Teile
    xIN_RestartCYCL : BOOL;          // Zyklus erneut starten im STEP: END: LEERFAHREN
    enIN_State      : enState;       // Status Anlage
    tIN_Timeout     : TIME := T#10s; // Timout

    pxFG_Freigabe : POINTER TO BOOL; //Freigabe von Station

    // Application specific
    Mover : REFERENCE TO FB_Mover;
END_VAR
VAR_OUTPUT
    (* standart Ausgänge *)
    xOUT_ErrFlag  : BOOL;         // Error Flag 
    xOUT_Busy     : BOOL;         // Baustein befindet sich im Ablauf 
    xOUT_Done     : BOOL;         // Baustein hat den Ablauf beendet 		
    xOUT_Ready    : BOOL;         // Ready to begin: should be the same state as done	
    xOUT_Timeout  : BOOL;         // Timeout FB 
    xOUT_InitDone : BOOL;         // initialisierung fertig
    xOUT_Wait     : BOOL;         // Wartet auf Bedingung
    iOUT_Step     : ST130_Dose_e; // Aktueller Schritt 
    sOUT_Step     : STRING;       // Aktueller Schritt but in string format
    bOUT_Error    : BYTE;         // Fehlernummer

    iOUT_ProcessCompletion : INT;  //process completion: express in % (0-100)
    xOUT_MoverFree         : BOOL; // The mover is free to move

END_VAR
VAR
    (* Standard *)
    (* Schritt *)
    iLastStep : ST130_Dose_e; // Merker letzter Schritt 
    iPreStep  : ST130_Dose_e; // Schritt zurück nach Alarm 
    iAktStep  : ST130_Dose_e; // aktueller Schritt

    // Trigger Starten 
    rtSTART : R_TRIG;
    // Timer TimeOut 
    TON_Timeout : TON;

    (* Bausteine *)

    (* Spezial *)
    fb_axis130_01Z : FB_AxisLIN_V1_1;
    fb_axis130_10Z : FB_AxisLM_V1_1;

    fb_VerAxis_01 : FB_LinearMotionMan;
    fb_VerAxis_10 : FB_LinearMotionMan;

    fb_simu_axis130_01Z : FB_Simu_AxisLIN_V1_1;
    fb_simu_axis130_10Z : FB_Simu_AxisLM_V1_1;

    // pneumatics
    fb_Kammer_Offnen_Links      : FB_ZylMo2El_V2_1;
    fb_Kammer_Offnen_Rechts     : FB_ZylMo2El_V2_1;
    fb_Kammer_nachfullen_Links  : FB_ZylMo2El_V2_1;
    fb_Kammer_nachfullen_Rechts : FB_ZylMo2El_V2_1;
    fb_Niederhalter_Patrone     : FB_ZylMo2El_V2_1;

    simu_Kammer_Offnen_Links      : FB_Simu_Zyl2Pos;
    simu_Kammer_Offnen_Rechts     : FB_Simu_Zyl2Pos;
    simu_Kammer_nachfullen_Links  : FB_Simu_Zyl2Pos;
    simu_Kammer_nachfullen_Rechts : FB_Simu_Zyl2Pos;
    simu_Niederhalter_Patrone     : FB_Simu_Zyl2Pos;

    fb_viebrieren_kammer_links  : FB_ZylMo2El_V2_1;
    fb_viebrieren_kammer_rechts : FB_ZylMo2El_V2_1;

    TON_load_kammer  : TON;
    TON_load_patrone : TON;

END_VAR
VAR CONSTANT
    DOSE_SIMULATION : BOOL := FALSE; // Set to TRUE to simulate this part of the program
END_VAR

(*******************************************************************)
(* Trigger  *)
(*******************************************************************)
(* Zurücksetzen *)
IF xIN_RESET THEN
    iPreStep  := ST130_Dose_e.RESET;
    iOUT_Step := ST130_Dose_e.RESET;
END_IF;

(* Error Quittieren *)
IF (bOUT_Error <> 0) AND xIN_Quit THEN
    xOUT_ErrFlag := FALSE;
    bOUT_Error   := 0;
    iOUT_Step    := iPreStep;
END_IF;

(*******************************************************************)
(* Timer *)
(*******************************************************************)
TON_Timeout(IN := xIN_NextStep AND (iLastStep = iOUT_Step) (*todo FG *) ,
            PT := tIN_Timeout);

TON_load_kammer(IN := ST130_Dose_e.fill_kammer = iOUT_Step,
                PT := DINT_TO_TIME(_20_AUTO.recipe.st130.diLoadKammer_ms));

TON_load_patrone(IN := ST130_Dose_e.load_powder_and_vibrate = iOUT_Step,
                 PT := DINT_TO_TIME(_20_AUTO.recipe.st130.diLoadPatrone_ms));

(*******************************************************************)
(* Bausteine *)
(*******************************************************************)
fb_VerAxis_01(config          := _20_AUTO.recipe.linearAxis[LinearAxis_e.ST130_01Z],
              xIN_Init        := enIN_State = enState.StateINIT,
              xIN_Reset       := xIN_Reset,
              lrIN_CurrPos    := fb_axis130_01Z.rOUT_ActPos,
              lrIN_Delta_mm   := 0.05,
              iIN_CurrentStep := iOUT_Step,
              iIN_moveNumber  := ST130_DosierkammerPos_e._max);

fb_simu_axis130_01Z(xIN_InSimu    := DOSE_SIMULATION AND CONST.USE_SIMULATION,
                    pIN_axisSimu  := ADR(SIMU.axis_ref[Axis_e.ST130_01Z]),
                    pIN_axisHW    := ADR(ST130_Axis.axis130_01Z.axis),
                    rIN_PosActual := ST130_Axis.axis130_01Z.rActPos,
                    rIN_PosMax    := ST130_Axis.const130_01Z.POS_MAX,
                    rIN_PosMin    := ST130_Axis.const130_01Z.POS_MIN,
                    rIN_PixMax    := 60,
                    rIN_PixMin    := 0);

// **** adjuste position
fb_axis130_01Z.rIN_Position := TO_REAL(fb_VerAxis_01.OUT_MoveProfile.lrPosition);

IF ST130_Dose_e.Adjust_Vertical_01Z_position = iOUT_Step THEN
    fb_axis130_01Z.rIN_Position := fb_axis130_01Z.rIN_Position + GVL.ST130_01Y_Feedback_Offset;
END_IF
// **** END adjuste position

fb_axis130_01Z(enIN_State      := enIN_State,
               parIN_Buttons   := ADR(AXIS.btTeachArAxis[Axis_e.ST130_01Z]),
               xIN_DisButtons  := FALSE,
               xIN_Quit        := xIN_Quit,
               xIN_AX5000      := FALSE,
               xIN_ENC_ABS     := TRUE,
               xIN_PARAMok     := TRUE,
               xIN_FREE        := TRUE,
               xIN_FREE_HOME   := TRUE,
               rIN_POSMIN      := ST130_Axis.const130_01Z.POS_MIN,
               rIN_POSMAX      := ST130_Axis.const130_01Z.POS_MAX,
               rIN_VELOMAX     := ST130_Axis.const130_01Z.VELO_MAX,
               rIN_VELOMANU    := ST130_Axis.const130_01Z.VELO_MANU,
               rIN_VELOOPEN    := ST130_Axis.const130_01Z.VELO_MANU / 4,
               rIN_JogInc      := AXIS.rTeachIncAxis,
               rIN_VeloJogManu := TO_REAL(AXIS.rJogVelo_pc),
               rIN_PosManu     := TO_REAL(_20_AUTO.recipe.linearAxis[LinearAxis_e.ST130_01Z]
                                              .movesList[AXIS.bTeachPos[Axis_e.ST130_01Z]].lrPosition),
               xIN_HomeExe      := FALSE,
               xIN_HomeCalib    := FALSE,
               xIN_Execute      := fb_VerAxis_01.xOUT_Execute,
               xIN_Relative     := FALSE,
               rIN_Position     :=, // set above due to automatic adjustement from GVL
               rIN_Velocity     := TO_REAL(fb_VerAxis_01.OUT_MoveProfile.lrVelocity),
               rIN_Acceleration := TO_REAL(fb_VerAxis_01.OUT_MoveProfile.lrAccel),
               rIN_Deceleration := TO_REAL(fb_VerAxis_01.OUT_MoveProfile.lrDecel),
               rIN_Jerk         := TO_REAL(fb_VerAxis_01.OUT_MoveProfile.lrJerk),
               xIN_Reset        := xIN_Reset,
               rOUT_ActPos      => ST130_Axis.axis130_01Z.rActPos,
               axisIN_REF       := fb_simu_axis130_01Z.pOUT_axisRef^);

fb_VerAxis_10(config          := _20_AUTO.recipe.linearAxis[LinearAxis_e.ST130_10Z],
              xIN_Init        := enIN_State = enState.StateINIT,
              xIN_Reset       := xIN_Reset,
              lrIN_CurrPos    := fb_axis130_10Z.rOUT_ActPos,
              lrIN_Delta_mm   := 1.0,
              iIN_CurrentStep := iOUT_Step,
              iIN_moveNumber  := ST130_PatroneAushebenPos_e._max);

fb_simu_axis130_10Z(xIN_Enable          := DOSE_SIMULATION AND CONST.USE_SIMULATION,
                    bIN_AxisCntr        := fb_axis130_10Z.bOUT_AxisCntr,
                    wIN_AxisState       := ST130_Axis.axis130_10Z.wState,
                    udiIN_HomingTime_ms := 2000,
                    pIN_axisSimu        := ADR(SIMU.axis_ref[Axis_e.ST130_10Z]),
                    pIN_axisHW          := ADR(ST130_Axis.axis130_10Z.axis),
                    rIN_PosActual       := ST130_Axis.axis130_10Z.rActPos,
                    rIN_PosMax          := ST130_Axis.const130_10Z.POS_MAX,
                    rIN_PosMin          := ST130_Axis.const130_10Z.POS_MIN,
                    rIN_PixMax          := 100,
                    rIN_PixMin          := 0);

fb_axis130_10Z(enIN_State       := enIN_State,
               parIN_Buttons    := ADR(AXIS.btTeachArAxis[Axis_e.ST130_10Z]),
               xIN_DisButtons   := FALSE,
               xIN_Quit         := xIN_Quit,
               xIN_PARAMok      := TRUE,
               xIN_FREE         := TRUE,
               xIN_FREE_HOME    := TRUE,
               rIN_POSMIN       := ST130_Axis.const130_10Z.POS_MIN,
               rIN_POSMAX       := ST130_Axis.const130_10Z.POS_MAX,
               rIN_VELOMAX      := ST130_Axis.const130_10Z.VELO_MAX,
               rIN_VELOMANU     := ST130_Axis.const130_10Z.VELO_MANU,
               rIN_VELOOPEN     := ST130_Axis.const130_10Z.POS_MAX / 4,
               rIN_JogInc       := AXIS.rTeachIncAxis,
               xIN_Execute      := fb_VerAxis_10.xOUT_Execute,
               xIN_Relative     := FALSE,
               xIN_STOP         := FALSE,
               xIN_OFF          := FALSE,
               rIN_Position     := TO_REAL(fb_VerAxis_10.OUT_MoveProfile.lrPosition),
               rIN_Velocity     := TO_REAL(fb_VerAxis_10.OUT_MoveProfile.lrVelocity),
               rIN_Acceleration := TO_REAL(fb_VerAxis_10.OUT_MoveProfile.lrAccel),
               rIN_Deceleration := TO_REAL(fb_VerAxis_10.OUT_MoveProfile.lrDecel),
               rIN_Jerk         := TO_REAL(fb_VerAxis_10.OUT_MoveProfile.lrJerk),
               rIN_PosManu      := TO_REAL(_20_AUTO.recipe.linearAxis[LinearAxis_e.ST130_10Z]
                                               .movesList[AXIS.bTeachPos[Axis_e.ST130_10Z]].lrPosition),
               rIN_VeloJogManu := TO_REAL(Axis.rJogVelo_pc),
               xIN_Home        := ST130_Dose_e.Init_HomeVertical_10 = iOUT_Step,
               xIN_Reset       := (ST130_Dose_e.RESET = iOUT_Step) OR xIN_Reset,
               wAxisState      := fb_simu_axis130_10Z.wOUT_AxisState,
               bOUT_AxisCntr   => ST130_Axis.axis130_10Z.bCtrlHi,
               rOUT_ActPos     => ST130_Axis.axis130_10Z.rActPos,
               axisIN_REF      := fb_simu_axis130_10Z.pOUT_axisRef^);

//////////////////////////////////
fb_Kammer_Offnen_Links(xIN_Reset    := xIN_Reset OR (ST130_Dose_e.RESET = iOUT_Step),
                       xIN_Quit     := xIN_Quit,
                       xIN_Manu     := enState.StateMANU = enIN_State,
                       pbtIN_Button := ADR(HMI.btManuCylinders[StationList_e.ST130][1]),
                       xIN_GS       := simu_Kammer_Offnen_Links.xOUT_inGS,
                       xIN_AS       := simu_Kammer_Offnen_Links.xOUT_inAS,
                       xIN_FREE     := TRUE,
                       xINtoGS      := ST130_Dose_e.Init_close_down_feeder = iOUT_Step OR
                                       ST130_Dose_e.close_down_feeder = iOUT_Step,
                       xINtoAS := _20_AUTO.recipe.st130.xUseVerLeft AND
                                  ST130_Dose_e.open_down_feeder = iOUT_Step,
                       tIN_ErrAS := DINT_TO_TIME(_20_AUTO.recipe.cylinder2Pos[StationList_e.ST130]
                                                     [ST130_Cylinders_e.Kammer_nachfullen_Links].toAS_alarm_time),
                       tIN_ErrGS := DINT_TO_TIME(_20_AUTO.recipe.cylinder2Pos[StationList_e.ST130]
                                                     [ST130_Cylinders_e.Kammer_Offnen_Links].toGS_alarm_time),
                       tIN_WaitAS := DINT_TO_TIME(_20_AUTO.recipe.cylinder2Pos[StationList_e.ST130]
                                                      [ST130_Cylinders_e.Kammer_Offnen_Links].toAS_wait_time),
                       tIN_WaitGS := DINT_TO_TIME(_20_AUTO.recipe.cylinder2Pos[StationList_e.ST130]
                                                      [ST130_Cylinders_e.Kammer_Offnen_Links].toGS_wait_time));

simu_Kammer_Offnen_Links(xIN_Enable := DOSE_SIMULATION AND CONST.USE_SIMULATION,
                         xIN_inGS   := IO_BOX.I1405_ST130_kammer_offnen_links_vor,
                         xIN_inAS   := IO_BOX.I1404_ST130_kammer_offnen_links_zuruck,
                         xIN_valve  := fb_Kammer_Offnen_Links.xOUT_VALVE,
                         tIN_GS_ms  := 200,  //ms
                         tIN_AS_ms  := 200); //ms

fb_Kammer_Offnen_Rechts(xIN_Reset    := xIN_Reset OR (ST130_Dose_e.RESET = iOUT_Step),
                        xIN_Quit     := xIN_Quit,
                        xIN_Manu     := enState.StateMANU = enIN_State,
                        pbtIN_Button := ADR(HMI.btManuCylinders[StationList_e.ST130][2]),
                        xIN_GS       := simu_Kammer_Offnen_Rechts.xOUT_inGS,
                        xIN_AS       := simu_Kammer_Offnen_Rechts.xOUT_inAS,
                        xIN_FREE     := TRUE,
                        xINtoGS      := ST130_Dose_e.Init_close_down_feeder = iOUT_Step OR
                                        ST130_Dose_e.close_down_feeder = iOUT_Step,
                        xINtoAS := _20_AUTO.recipe.st130.xUseVerRight AND
                                   ST130_Dose_e.open_down_feeder = iOUT_Step,
                        tIN_ErrAS := DINT_TO_TIME(_20_AUTO.recipe.cylinder2Pos[StationList_e.ST130]
                                                      [ST130_Cylinders_e.Kammer_Offnen_Rechts].toAS_alarm_time),
                        tIN_ErrGS := DINT_TO_TIME(_20_AUTO.recipe.cylinder2Pos[StationList_e.ST130]
                                                      [ST130_Cylinders_e.Kammer_Offnen_Rechts].toGS_alarm_time),
                        tIN_WaitAS := DINT_TO_TIME(_20_AUTO.recipe.cylinder2Pos[StationList_e.ST130]
                                                       [ST130_Cylinders_e.Kammer_Offnen_Rechts].toAS_wait_time),
                        tIN_WaitGS := DINT_TO_TIME(_20_AUTO.recipe.cylinder2Pos[StationList_e.ST130]
                                                       [ST130_Cylinders_e.Kammer_Offnen_Rechts].toGS_wait_time));

simu_Kammer_Offnen_Rechts(xIN_Enable := DOSE_SIMULATION AND CONST.USE_SIMULATION,
                          xIN_inGS   := IO_BOX.I1407_ST130_kammer_offnen_rechts_vor,
                          xIN_inAS   := IO_BOX.I1406_ST130_kammer_offnen_rechts_zuruck,
                          xIN_valve  := fb_Kammer_Offnen_Rechts.xOUT_VALVE,
                          tIN_GS_ms  := 200,  //ms
                          tIN_AS_ms  := 200); //ms

fb_Kammer_nachfullen_Links(xIN_Reset    := xIN_Reset OR (ST130_Dose_e.RESET = iOUT_Step),
                           xIN_Quit     := xIN_Quit,
                           xIN_Manu     := enState.StateMANU = enIN_State,
                           pbtIN_Button := ADR(HMI.btManuCylinders[StationList_e.ST130][3]),
                           xIN_GS       := simu_Kammer_nachfullen_Links.xOUT_inGS,
                           xIN_AS       := simu_Kammer_nachfullen_Links.xOUT_inAS,
                           xIN_FREE     := TRUE,
                           xINtoGS      := (ST130_Dose_e.close_up_feeder = iOUT_Step) OR
                                           (ST130_Dose_e.Init_close_up_feeder = iOUT_Step) OR
                                           (enIN_State < enState.StateSTEP),
                           xINtoAS := _20_AUTO.recipe.st130.xUseVerLeft AND
                                      (enIN_State >= enState.StateSTEP) AND
                                      (ST130_Dose_e.open_up_feeder = iOUT_Step OR
                                      ST130_Dose_e.open_up_feeder_first = iOUT_Step),
                           tIN_ErrAS := DINT_TO_TIME(_20_AUTO.recipe.cylinder2Pos[StationList_e.ST130]
                                                         [ST130_Cylinders_e.Kammer_nachfullen_Links]
                                                         .toAS_alarm_time),
                           tIN_ErrGS := DINT_TO_TIME(_20_AUTO.recipe.cylinder2Pos[StationList_e.ST130]
                                                         [ST130_Cylinders_e.Kammer_nachfullen_Links].toGS_alarm_time),
                           tIN_WaitAS := DINT_TO_TIME(_20_AUTO.recipe.cylinder2Pos[StationList_e.ST130]
                                                          [ST130_Cylinders_e.Kammer_nachfullen_Links].toAS_wait_time),
                           tIN_WaitGS := DINT_TO_TIME(_20_AUTO.recipe.cylinder2Pos[StationList_e.ST130]
                                                          [ST130_Cylinders_e.Kammer_nachfullen_Links].toGS_wait_time));

simu_Kammer_nachfullen_Links(xIN_Enable := DOSE_SIMULATION AND CONST.USE_SIMULATION,
                             xIN_inGS   := IO_BOX.I1400_ST130_nachfullen_offnen_links_zuruck,
                             xIN_inAS   := IO_BOX.I1401_ST130_nachfullen_offnen_links_vor,
                             xIN_valve  := fb_Kammer_nachfullen_Links.xOUT_VALVE,
                             tIN_GS_ms  := 200,  //ms
                             tIN_AS_ms  := 200); //ms

fb_Kammer_nachfullen_Rechts(xIN_Reset    := xIN_Reset OR (ST130_Dose_e.RESET = iOUT_Step),
                            xIN_Quit     := xIN_Quit,
                            xIN_Manu     := enState.StateMANU = enIN_State,
                            pbtIN_Button := ADR(HMI.btManuCylinders[StationList_e.ST130][4]),
                            xIN_GS       := simu_Kammer_nachfullen_Rechts.xOUT_inGS,
                            xIN_AS       := simu_Kammer_nachfullen_Rechts.xOUT_inAS,
                            xIN_FREE     := TRUE,
                            xINtoGS      := (ST130_Dose_e.close_up_feeder = iOUT_Step) OR
                                            (ST130_Dose_e.Init_close_up_feeder = iOUT_Step) OR
                                            (enIN_State < enState.StateSTEP),
                            xINtoAS := _20_AUTO.recipe.st130.xUseVerRight AND
                                       (enIN_State >= enState.StateSTEP) AND
                                       (ST130_Dose_e.open_up_feeder = iOUT_Step OR
                                       ST130_Dose_e.open_up_feeder_first = iOUT_Step),
                            tIN_ErrAS := DINT_TO_TIME(_20_AUTO.recipe.cylinder2Pos[StationList_e.ST130]
                                                          [ST130_Cylinders_e.Kammer_nachfullen_Rechts]
                                                          .toAS_alarm_time),
                            tIN_ErrGS := DINT_TO_TIME(_20_AUTO.recipe.cylinder2Pos[StationList_e.ST130]
                                                          [ST130_Cylinders_e.Kammer_nachfullen_Rechts]
                                                          .toGS_alarm_time),
                            tIN_WaitAS := DINT_TO_TIME(_20_AUTO.recipe.cylinder2Pos[StationList_e.ST130]
                                                           [ST130_Cylinders_e.Kammer_nachfullen_Rechts]
                                                           .toAS_wait_time),
                            tIN_WaitGS := DINT_TO_TIME(_20_AUTO.recipe.cylinder2Pos[StationList_e.ST130]
                                                           [ST130_Cylinders_e.Kammer_nachfullen_Rechts]
                                                           .toGS_wait_time));

simu_Kammer_nachfullen_Rechts(xIN_Enable := DOSE_SIMULATION AND CONST.USE_SIMULATION,
                              xIN_inGS   := IO_BOX.I1402_ST130_nachfullen_offnen_rechts_zuruck,
                              xIN_inAS   := IO_BOX.I1403_ST130_nachfullen_offnen_rechts_vor,
                              xIN_valve  := fb_Kammer_nachfullen_Rechts.xOUT_VALVE,
                              tIN_GS_ms  := 200,  // ms
                              tIN_AS_ms  := 200); // ms

fb_viebrieren_kammer_links(xIN_Reset    := xIN_Reset OR (ST130_Dose_e.RESET = iOUT_Step),
                           xIN_Quit     := xIN_Quit,
                           xIN_Manu     := enState.StateMANU = enIN_State,
                           pbtIN_Button := ADR(HMI.btManuCylinders[StationList_e.ST130][5]),
                           xIN_GS       := NOT fb_viebrieren_kammer_links.xOUT_VALVE, // no sensor here
                           xIN_AS       := fb_viebrieren_kammer_links.xOUT_VALVE,     // no sensor here
                           xIN_FREE     := TRUE,
                           xINtoGS      := NOT fb_viebrieren_kammer_links.xINtoAS,
                           xINtoAS      := _20_AUTO.recipe.st130.xUseVerLeft AND
                                           ((ST130_Dose_e.check_filterhut_presence <= iOUT_Step AND
                                           ST130_Dose_e.load_powder_and_vibrate >= iOUT_Step) OR
                                           (ST130_Dose_e.fill_kammer = iOUT_Step)),
                           tIN_ErrAS := DINT_TO_TIME(_20_AUTO.recipe.cylinder2Pos[StationList_e.ST130]
                                                         [ST130_Cylinders_e.Vibrieren_Kammer_Links]
                                                         .toAS_alarm_time),
                           tIN_ErrGS := DINT_TO_TIME(_20_AUTO.recipe.cylinder2Pos[StationList_e.ST130]
                                                         [ST130_Cylinders_e.Vibrieren_Kammer_Links]
                                                         .toGS_alarm_time),
                           tIN_WaitAS := DINT_TO_TIME(_20_AUTO.recipe.cylinder2Pos[StationList_e.ST130]
                                                          [ST130_Cylinders_e.Vibrieren_Kammer_Links]
                                                          .toAS_wait_time),
                           tIN_WaitGS := DINT_TO_TIME(_20_AUTO.recipe.cylinder2Pos[StationList_e.ST130]
                                                          [ST130_Cylinders_e.Vibrieren_Kammer_Links]
                                                          .toGS_wait_time));

fb_viebrieren_kammer_rechts(xIN_Reset    := xIN_Reset OR (ST130_Dose_e.RESET = iOUT_Step),
                            xIN_Quit     := xIN_Quit,
                            xIN_Manu     := enState.StateMANU = enIN_State,
                            pbtIN_Button := ADR(HMI.btManuCylinders[StationList_e.ST130][6]),
                            xIN_GS       := NOT fb_viebrieren_kammer_rechts.xOUT_VALVE, // no sensor here
                            xIN_AS       := fb_viebrieren_kammer_rechts.xOUT_VALVE,     // no sensor here
                            xIN_FREE     := TRUE,
                            xINtoGS      := NOT fb_viebrieren_kammer_links.xINtoAS,
                            xINtoAS      := _20_AUTO.recipe.st130.xUseVerRight AND
                                            ((ST130_Dose_e.check_filterhut_presence <= iOUT_Step AND
                                            ST130_Dose_e.load_powder_and_vibrate >= iOUT_Step) OR
                                            (ST130_Dose_e.fill_kammer = iOUT_Step)),
                            tIN_ErrAS := DINT_TO_TIME(_20_AUTO.recipe.cylinder2Pos[StationList_e.ST130]
                                                          [ST130_Cylinders_e.Vibrieren_Kammer_Rechts]
                                                          .toAS_alarm_time),
                            tIN_ErrGS := DINT_TO_TIME(_20_AUTO.recipe.cylinder2Pos[StationList_e.ST130]
                                                          [ST130_Cylinders_e.Vibrieren_Kammer_Rechts]
                                                          .toGS_alarm_time),
                            tIN_WaitAS := DINT_TO_TIME(_20_AUTO.recipe.cylinder2Pos[StationList_e.ST130]
                                                           [ST130_Cylinders_e.Vibrieren_Kammer_Rechts]
                                                           .toAS_wait_time),
                            tIN_WaitGS := DINT_TO_TIME(_20_AUTO.recipe.cylinder2Pos[StationList_e.ST130]
                                                           [ST130_Cylinders_e.Vibrieren_Kammer_Rechts]
                                                           .toGS_wait_time));

fb_Niederhalter_Patrone(xIN_Reset    := xIN_Reset OR (ST130_Dose_e.RESET = iOUT_Step),
                        xIN_Quit     := xIN_Quit,
                        xIN_Manu     := enState.StateMANU = enIN_State,
                        pbtIN_Button := ADR(HMI.btManuCylinders[StationList_e.ST130][7]),
                        xIN_GS       := simu_Niederhalter_Patrone.xOUT_inGS,
                        xIN_AS       := simu_Niederhalter_Patrone.xOUT_inAS,
                        xIN_FREE     := TRUE,
                        xINtoGS      := ST130_Dose_e.Init_clamp_up = iOUT_Step OR
                                        ST130_Dose_e.clamp_up = iOUT_Step,
                        xINtoAS   := ST130_Dose_e.clamp_down = iOUT_Step,
                        tIN_ErrAS := DINT_TO_TIME(_20_AUTO.recipe.cylinder2Pos[StationList_e.ST130]
                                                      [ST130_Cylinders_e.Niederhalter_Patrone]
                                                      .toAS_alarm_time),
                        tIN_ErrGS := DINT_TO_TIME(_20_AUTO.recipe.cylinder2Pos[StationList_e.ST130]
                                                      [ST130_Cylinders_e.Niederhalter_Patrone]
                                                      .toGS_alarm_time),
                        tIN_WaitAS := DINT_TO_TIME(_20_AUTO.recipe.cylinder2Pos[StationList_e.ST130]
                                                       [ST130_Cylinders_e.Niederhalter_Patrone]
                                                       .toAS_wait_time),
                        tIN_WaitGS := DINT_TO_TIME(_20_AUTO.recipe.cylinder2Pos[StationList_e.ST130]
                                                       [ST130_Cylinders_e.Niederhalter_Patrone]
                                                       .toGS_wait_time));

simu_Niederhalter_Patrone(xIN_Enable := DOSE_SIMULATION AND CONST.USE_SIMULATION,
                          xIN_inGS   := IO_BOX.I2100_ST130_niederhalter_patrone_oben,
                          xIN_inAS   := IO_BOX.I2101_ST130_niederhalter_patrone_unten,
                          xIN_valve  := fb_Niederhalter_Patrone.xOUT_VALVE,
                          tIN_GS_ms  := 200,  // ms
                          tIN_AS_ms  := 200); // ms

(*******************************************************************)
(* OUTPUTS *)
(*******************************************************************)
// Error Flag 
xOUT_ErrFlag := (bOUT_Error <> 0) OR (ST130_Dose_e.ERROR = iOUT_Step);
// Baustein befindet sich im Ablauf 
xOUT_Busy := (iOUT_Step > ST130_Dose_e.READY) AND (iOUT_Step < ST130_Dose_e.DONE);
// Baustein hat den Ablauf beendet
xOUT_Done := (iOUT_Step = ST130_Dose_e.DONE);
// Process ready
xOUT_Ready := (iOUT_Step = ST130_Dose_e.READY) OR (iOUT_Step = ST130_Dose_e.waitOnMover);
// Timeout FB 				 		
xOUT_Timeout := TON_Timeout.Q;
// Itialisierung fertig			
xOUT_InitDone := (iOUT_Step = ST130_Dose_e.READY) OR
                 (iOUT_Step = ST130_Dose_e.waitOnMover) OR
                 (iOUT_Step = ST130_Dose_e.DONE);

// Aktueller Schritt			
iOUT_Step := iOUT_Step; //Im Ablauf gesetzt		
sOUT_Step := TO_STRING(iOUT_Step);
//Fehlernummer	 
bOUT_Error := bOUT_Error; //Im Ablauf/FB gesetzt	
(* Warte (alle Schritte wo auf FG oder Teile gewartet wird) *)
xOUT_Wait := (iOUT_Step = ST130_Dose_e.DONE) OR
             (iOUT_Step = ST130_Dose_e.READY) OR
             (iOUT_Step = ST130_Dose_e.START) OR
             (iOUT_Step = ST130_Dose_e.waitOnMover) OR
             (iOUT_Step = ST130_Dose_e.SYNC_MOVER_LEAVE);

xOUT_MoverFree :=
    NOT (iOUT_Step >= ST130_Dose_e.MOVER_NEEDED_OP AND iOUT_Step < ST130_Dose_e.MOVER_FREE_OP) AND
    (iOUT_Step >= ST130_Dose_e.READY) AND
    (iOUT_Step < ST130_Dose_e.ERROR);

iOUT_ProcessCompletion := F_GetPercent_2(iOUT_Step,
                                         ST130_Dose_e.waitOnMover,
                                         ST130_Dose_e.DONE,
                                         ST130_Dose_e.waitOnMover,
                                         ST130_Dose_e.DONE);

IO_BOX.Q0100_14_ST130_kammer_offnen_links :=
    fb_Kammer_Offnen_Links.xOUT_VALVE AND
    NOT IO_BOX.Q0102_14_ST130_kammer_nachfullen_links AND
    ((enIN_State >= enState.StateALARM) AND // we must ensure that kammer is closed when not in automatic mode
    (NOT (DOSE_SIMULATION AND CONST.USE_SIMULATION)) OR
    (enIN_State = enState.StateMANU));

IO_BOX.Q0101_14_ST130_kammer_offnen_rechts :=
    fb_Kammer_Offnen_Rechts.xOUT_VALVE AND
    NOT IO_BOX.Q0103_14_ST130_kammer_nachfullen_rechts AND
    ((enIN_State >= enState.StateALARM) AND // we must ensure that kammer is closed when not in automatic mode
    (NOT (DOSE_SIMULATION AND CONST.USE_SIMULATION)) OR
    (enIN_State = enState.StateMANU));

IO_BOX.Q0102_14_ST130_kammer_nachfullen_links :=
    fb_Kammer_nachfullen_Links.xOUT_VALVE AND
    ((enIN_State >= enState.StateALARM) AND // we must ensure that kammer is closed when not in automatic mode
    (NOT (DOSE_SIMULATION AND CONST.USE_SIMULATION)) OR
    (enIN_State = enState.StateMANU));

IO_BOX.Q0103_14_ST130_kammer_nachfullen_rechts :=
    fb_Kammer_nachfullen_Rechts.xOUT_VALVE AND
    ((enIN_State >= enState.StateALARM) AND // we must ensure that kammer is closed when not in automatic mode
    (NOT (DOSE_SIMULATION AND CONST.USE_SIMULATION)) OR
    (enIN_State = enState.StateMANU));

IO_BOX.Q0104_14_ST130_vibrieren_kammer_links :=
    fb_viebrieren_kammer_links.xOUT_VALVE AND
    (NOT (DOSE_SIMULATION AND CONST.USE_SIMULATION) OR (enIN_State = enState.StateMANU));

IO_BOX.Q0104_12_ST130_vibrieren_kammer_rechts :=
    fb_viebrieren_kammer_rechts.xOUT_VALVE AND
    (NOT (DOSE_SIMULATION AND CONST.USE_SIMULATION) OR (enIN_State = enState.StateMANU));

IO_BOX.Q0105_14_ST130_niederhalter_patrone :=
    fb_Niederhalter_Patrone.xOUT_VALVE AND
    (NOT (DOSE_SIMULATION AND CONST.USE_SIMULATION) OR (enIN_State = enState.StateMANU));

_20_AUTO.recipe.st130.uiVibroUnderneath := LIMIT(UINT#0, _20_AUTO.recipe.st130.uiVibroUnderneath, UINT#100);

IF IO_BOX.Q0104_14_ST130_vibrieren_kammer_links AND (ST130_Dose_e.fill_kammer <> iOUT_Step) THEN
    OUT.QA01_ST130_pressure_valve_left := (UINT#16#FFFF / UINT#100) * _20_AUTO.recipe.st130.uiVibroUnderneath;
ELSE
    OUT.QA01_ST130_pressure_valve_left := 0;
END_IF

IF IO_BOX.Q0104_12_ST130_vibrieren_kammer_rechts AND (ST130_Dose_e.fill_kammer <> iOUT_Step) THEN
    OUT.QA02_ST130_pressure_valve_right := (UINT#16#FFFF / UINT#100) * _20_AUTO.recipe.st130.uiVibroUnderneath;
ELSE
    OUT.QA02_ST130_pressure_valve_right := 0;
END_IF

(*******************************************************************)
(* Ablauf *)
(*******************************************************************)

(* Sperren *)
IF xIN_Sperre THEN
    iPreStep  := ST130_Dose_e.RESET;
    iOUT_Step := ST130_Dose_e.RESET;
    RETURN;
END_IF;

(* Schritt Merker *)
IF iAktStep <> iOUT_Step THEN
    iLastStep := iAktStep;
    iAktStep  := iOUT_Step;
END_IF

(* START *)
rtSTART(CLK := xIN_Start);

IF 0 = bOUT_Error THEN
    IF fb_axis130_01Z.xOUT_ErrFlag THEN
        bOUT_Error := 11;
    ELSIF fb_axis130_10Z.xOUT_ErrFlag THEN
        bOUT_Error := 12;
    ELSIF fb_Kammer_Offnen_Links.xOUT_ErrFlag THEN
        bOUT_Error := 20;
    ELSIF fb_Kammer_Offnen_Rechts.xOUT_ErrFlag THEN
        bOUT_Error := 21;
    ELSIF fb_Kammer_nachfullen_Links.xOUT_ErrFlag THEN
        bOUT_Error := 22;
    ELSIF fb_Kammer_nachfullen_Rechts.xOUT_ErrFlag THEN
        bOUT_Error := 23;
    ELSIF fb_Niederhalter_Patrone.xOUT_ErrFlag THEN
        bOUT_Error := 24;
    ELSIF fb_viebrieren_kammer_links.xOUT_ErrFlag THEN
        bOUT_Error := 25;
    ELSIF fb_viebrieren_kammer_rechts.xOUT_ErrFlag THEN
        bOUT_Error := 26;
    END_IF
ELSIF iOUT_Step < ST130_Dose_e.ERROR THEN
    iOUT_Step := ST130_Dose_e.ERROR;
END_IF

(*******************************************************************)
(* Schrittkette  *)
(*******************************************************************)
CASE iOUT_Step OF

(***** RESET *****)
ST130_Dose_e.RESET: (* Schritt 0-99 *)
    //Initialisierungen
    //Start Init Ablauf
    IF xIN_Init THEN
        iOUT_Step := ST130_Dose_e.INIT;
        //Start Manu Ablauf
    ELSIF enIN_State = StateMANU AND xIN_NextStep THEN
        iOUT_Step := ST130_Dose_e.INIT;
    END_IF;

(***** INIT *****)
ST130_Dose_e.INIT: (* Grundstellung ? *)
    iOUT_Step := ST130_Dose_e.Init_Vertical_01Z_at_position;

ST130_Dose_e.Init_Vertical_01Z_at_position:
    IF fb_VerAxis_01.MoveTo(ST130_DosierkammerPos_e.down_AS).xOUT_InPos THEN
        IF fb_axis130_10Z.xOUT_HOMED THEN
            iOUT_Step := ST130_Dose_e.Init_Vertical_10_Down;
        ELSE
            iOUT_Step := ST130_Dose_e.Init_HomeVertical_10;
        END_IF
    END_IF

ST130_Dose_e.Init_HomeVertical_10:
    IF fb_axis130_10Z.xOUT_HOMED THEN
        iOUT_Step := ST130_Dose_e.Init_Vertical_10_Down;
    END_IF

ST130_Dose_e.Init_Vertical_10_Down:
    IF fb_VerAxis_10.MoveTo(ST130_PatroneAushebenPos_e.down_GS).xOUT_InPos THEN
        iOUT_Step := ST130_Dose_e.Init_close_down_feeder;
    END_IF

ST130_Dose_e.Init_close_down_feeder:
    IF (NOT _20_AUTO.recipe.st130.xUseVerLeft OR fb_Kammer_Offnen_Links.xOUT_inGS) AND
       (NOT _20_AUTO.recipe.st130.xUseVerRight OR fb_Kammer_Offnen_Rechts.xOUT_inGS) THEN
        iOUT_Step := ST130_Dose_e.Init_close_up_feeder;
    END_IF

ST130_Dose_e.Init_close_up_feeder:
    IF (NOT _20_AUTO.recipe.st130.xUseVerLeft OR fb_Kammer_nachfullen_Links.xOUT_inGS) AND
       (NOT _20_AUTO.recipe.st130.xUseVerRight OR fb_Kammer_nachfullen_Rechts.xOUT_inGS) THEN
        iOUT_Step := ST130_Dose_e.Init_clamp_up;
    END_IF

ST130_Dose_e.Init_clamp_up:
    IF fb_Niederhalter_Patrone.xOUT_inGS THEN
        iOUT_Step := ST130_Dose_e.READY;
    END_IF

(***** READY / INIT DONE *****)
ST130_Dose_e.READY:   (* Start AUTO:END:LEER:STEP *)
    IF xIN_Start THEN //IF rtSTART.Q THEN
        iOUT_Step := ST130_Dose_e.START;
    END_IF

(***** START  ZYKLISCH *****)
ST130_Dose_e.START: (*  *)
    IF xIN_NextStep AND pxFG_Freigabe^ THEN

        iPreStep := ST130_Dose_e.INIT;

        IF enState.StateLEER = enIN_State THEN
            IF __ISVALIDREF(Mover) THEN
                IF Mover.GetLastStationDone() > 0 THEN
                    iOUT_Step := ST130_Dose_e.Adjust_Vertical_01Z_position;
                ELSE
                    iOUT_Step := ST130_Dose_e.waitOnMover;
                END_IF
            END_IF
        ELSE
            iOUT_Step := ST130_Dose_e.open_up_feeder_first;
        END_IF
    END_IF;

ST130_Dose_e.Adjust_Vertical_01Z_position:
    IF xIN_NextStep AND
       fb_VerAxis_01.MoveTo(ST130_DosierkammerPos_e.down_AS).xOUT_InPos THEN
        iOUT_Step := ST130_Dose_e.open_up_feeder_first;
    END_IF

ST130_Dose_e.open_up_feeder_first:
    IF xIN_NextStep AND
       (NOT _20_AUTO.recipe.st130.xUseVerLeft OR fb_Kammer_nachfullen_Links.xOUT_inAS) AND
       (NOT _20_AUTO.recipe.st130.xUseVerRight OR fb_Kammer_nachfullen_Rechts.xOUT_inAS) THEN
        iOUT_Step := ST130_Dose_e.fill_kammer;
    END_IF

ST130_Dose_e.fill_kammer:
    IF xIN_NextStep AND TON_load_kammer.Q THEN
        iOUT_Step := ST130_Dose_e.waitOnMover;
    END_IF

ST130_Dose_e.waitOnMover:
    IF xIN_NextStep AND __ISVALIDREF(Mover) OR HMI.bArForceCyclusState[StationList_e.ST130] THEN
        IF Mover.GetLastStationDone() >= INT#130 THEN
            iOUT_Step := ST130_Dose_e.SYNC_MOVER_LEAVE;
        ELSIF Mover.GetLastStationDone() < INT#125 THEN
            iOUT_Step := ST130_Dose_e.SYNC_MOVER_LEAVE;
        ELSE
            iOUT_Step := ST130_Dose_e.check_filterhut_presence;
        END_IF
    END_IF

ST130_Dose_e.check_filterhut_presence:
    IF xIN_NextStep AND TRUE THEN
        iOUT_Step := ST130_Dose_e.close_up_feeder;
    END_IF

ST130_Dose_e.close_up_feeder:
    IF xIN_NextStep AND
       (NOT _20_AUTO.recipe.st130.xUseVerLeft OR fb_Kammer_nachfullen_Links.xOUT_inGS) AND
       (NOT _20_AUTO.recipe.st130.xUseVerRight OR fb_Kammer_nachfullen_Rechts.xOUT_inGS) THEN
        iOUT_Step := ST130_Dose_e.lift_up_piece_in_workposition;
    END_IF

ST130_Dose_e.lift_up_piece_in_workposition:
    IF xIN_NextStep AND fb_VerAxis_10.MoveTo(ST130_PatroneAushebenPos_e.up_AS).xOUT_InPos THEN
        IF DOSE_SIMULATION AND CONST.USE_SIMULATION THEN
            iOUT_Step := ST130_Dose_e.load_powder_and_vibrate;
        ELSE
            iOUT_Step := ST130_Dose_e.open_down_feeder;
        END_IF
    END_IF

ST130_Dose_e.open_down_feeder:
    IF xIN_NextStep AND
       (NOT _20_AUTO.recipe.st130.xUseVerLeft OR fb_Kammer_Offnen_Links.xOUT_inAS) AND
       (NOT _20_AUTO.recipe.st130.xUseVerRight OR fb_Kammer_Offnen_Rechts.xOUT_inAS) THEN
        iOUT_Step := ST130_Dose_e.load_powder_and_vibrate;

        IF __ISVALIDREF(Mover) THEN
            IF NOT Mover.SetLastStation(130) THEN
                ASSERT(0);
            END_IF
        END_IF
    END_IF

ST130_Dose_e.load_powder_and_vibrate:
    IF xIN_NextStep AND TON_load_patrone.Q THEN
        iOUT_Step := ST130_Dose_e.close_down_feeder;
    END_IF

ST130_Dose_e.close_down_feeder:
    IF xIN_NextStep AND
       (NOT _20_AUTO.recipe.st130.xUseVerLeft OR fb_Kammer_Offnen_Links.xOUT_inGS) AND
       (NOT _20_AUTO.recipe.st130.xUseVerRight OR fb_Kammer_Offnen_Rechts.xOUT_inGS) THEN
        iOUT_Step := ST130_Dose_e.release_piece_and_open_up_feeder;
    END_IF

ST130_Dose_e.release_piece_and_open_up_feeder:
    IF xIN_NextStep AND fb_VerAxis_10.MoveTo(ST130_PatroneAushebenPos_e.down_GS).xOUT_InPos THEN
        iOUT_Step := ST130_Dose_e.open_up_feeder;
    END_IF

ST130_Dose_e.open_up_feeder:
    IF xIN_NextStep AND
       (NOT _20_AUTO.recipe.st130.xUseVerLeft OR fb_Kammer_nachfullen_Links.xOUT_inAS) AND
       (NOT _20_AUTO.recipe.st130.xUseVerRight OR fb_Kammer_nachfullen_Rechts.xOUT_inAS) THEN
        iOUT_Step := ST130_Dose_e.clamp_down;
    END_IF

ST130_Dose_e.clamp_down:
    IF xIN_NextStep AND fb_Niederhalter_Patrone.xOUT_inAS THEN
        iOUT_Step := ST130_Dose_e.clamp_up;
    END_IF

ST130_Dose_e.clamp_up:
    IF xIN_NextStep AND fb_Niederhalter_Patrone.xOUT_inGS THEN
        iOUT_Step := ST130_Dose_e.SYNC_MOVER_LEAVE;

        IF __ISVALIDREF(Mover) THEN
            IF NOT Mover.SetLastStation(130) THEN
                ASSERT(0);
            END_IF
        END_IF
    END_IF

ST130_Dose_e.SYNC_MOVER_LEAVE:
    // The mover needs to be taken by MoverMan
    IF NOT __ISVALIDREF(Mover) THEN
        iOUT_Step := ST130_Dose_e.DONE;
    END_IF

(***** DONE *****)
ST130_Dose_e.DONE: (* Letzter Schritt  *)
    IF NOT xIN_AlarmAktiv THEN
        //AUTO
        IF (enIN_State = StateAUTO) AND xIN_RestartCYCL THEN
            iOUT_Step := ST130_Dose_e.START;
            //STEP / END / LEERFAHREN restart
        ELSIF (enIN_State < StateAUTO) AND (enIN_State >= enState.StateSTEP) AND xIN_RestartCYCL THEN
            iOUT_Step := ST130_Dose_e.START;
            //STEP / END / LEERFAHREN fertig
        ELSIF (enIN_State = StateREADY) THEN
            iOUT_Step := ST130_Dose_e.READY;
        END_IF;
    END_IF;

(************ ERROR *************)
ST130_Dose_e.ERROR: (* ERROR *) ;

END_CASE;

END_FUNCTION_BLOCK

// ---- POUs/20_AUTO/ST130/FB_AUT_135.TcPOU
FUNCTION_BLOCK FB_AUT_135 EXTENDS FB_AUT_ABSTRACT
(****************************************************************************)
(*	POU_AUT_zxx			Bausteinaufrufe Station	zxx							*)
(*	Status				ungetestet											*)
(*  Version:			1.0													*)
(*	Beschrieb:																*)
(*																			*)
(*	Abläufe:			FB_ABLzxxA		Hauptablauf							*)
(*																			*)
(*																			*)
(* 	25.09.2019/Dj															*)
(****************************************************************************)
(*	dd.mm.yyyy   KZ    x.y			Beschrieb								*)
(****************************************************************************)
VAR_INPUT
    (* spezifische Eingänge *)

END_VAR
VAR_OUTPUT
    (* spezifische Ausgänge *)

END_VAR
VAR
    (* Bausteine *)
    fb_Dose : FB_ABL_MODIFY_135;

    fb_stat : FB_AUT_Statistics;

END_VAR

(*******************************************************************)
(* Timer *)
(*******************************************************************)

(*******************************************************************)
(* Flanken / Merker *)
(*******************************************************************)
//MANU CYCLE
IF (enIN_State = StateMANU) AND xIN_ManuCycle THEN
    xManuCycle := TRUE;
END_IF;

IF (enIN_State <> StateMANU) OR xOUT_Done THEN
    xManuCycle := FALSE;
END_IF

//NEXT STEP
xNextStep := (enIN_State > StateSTEP) OR
             ((enIN_State = StateSTEP) AND xIN_Step) OR
             ((enIN_State = StateMANU) AND xManuCycle);

//RESET
xReset := (enIN_State < StateREADY) AND (enIN_State <> StateINIT) AND NOT xManuCycle;

(*******************************************************************)
(* Bausteinaufrufe Abläufe *)
(*******************************************************************)

xRelease := MAIN.MoverMan.IsProcessUsed(THIS^);

fb_Dose(xIN_Reset         := xReset,
        xIN_Init          := xIN_Init,
        xIN_Quit          := xIN_Quit,
        xIN_Start         := enIN_State >= enState.StateLEER, //AND _FB_ABL_100A.xOUT_Done AND _FB_ABL_100A.xOUT_Ready,
        xIN_Sperre        := NOT xIN_On,
        xIN_NextStep      := xNextStep,
        xIN_AlarmAktiv    := xIN_AlarmAktiv,
        xIN_DryCycle      := xIN_DryCycle,
        xIN_RestartCYCL   := enIN_State >= enState.StateLEER, // only restart when the mover has move out
        enIN_State        := enIN_State,
        tIN_Timeout       := tIN_Timeout,
        pxFG_Freigabe     := ADR(xRelease),
        Mover             := THIS^.Mover,
        iProcessTimeMili1 := DINT_TO_UDINT(THIS^.iProcessTimeMili_1),
        iProcessTimeMili2 := DINT_TO_UDINT(THIS^.iProcessTimeMili_2));

fb_stat(xIN_Enable  := enState.StateAUTO = enIN_State,
        xIN_Waiting := fb_Dose.xOUT_Wait,
        xIN_Running := (fb_Dose.iOUT_Step >= ST100_Modify_e.START) AND
                       (fb_Dose.iOUT_Step <= ST100_Modify_e.DONE),
        // Since we use a mover system, a cycle is done when we are waiting on a mover
        xIN_Done := fb_Dose.iOUT_Step = ST100_Modify_e.waitOnMover);

(*******************************************************************)
(* Mover reset flags *)
(*******************************************************************)

(*******************************************************************)
(* OUTPUT *)
(*******************************************************************)
xOUT_InitDone := fb_Dose.xOUT_InitDone;
xOUT_Ready    := fb_Dose.xOUT_Ready;
xOUT_Done     := fb_Dose.xOUT_Done;
xOUT_ErrFlag  := fb_Dose.xOUT_ErrFlag;
xOUT_Wait     := fb_Dose.xOUT_Wait;
xOUT_AlarmST  := xOUT_ErrFlag;

(*******************************************************************)
(* Bausteinaufruf Error Station *)
(*******************************************************************)
// POU_ERR_VORLAGE(xIN_QUIT:=xIN_Quit , pstrArIN_ALARM:=ADR(HMI.strArALARM[1]));

(* % of completion of the process *)
PROPERTY iCompletionPC : INT
GET
iCompletionPC := THIS^.fb_Dose.iOUT_ProcessCompletion;
END_GET
END_PROPERTY

(* Process time, expressed in milisecond *)
PROPERTY iProcessTimeMili_1 : DINT
GET
iProcessTimeMili_1 := TO_DINT(1000);
END_GET
END_PROPERTY

(* Process time, expressed in milisecond *)
PROPERTY iProcessTimeMili_2 : DINT
GET
iProcessTimeMili_2 := TO_DINT(1000);
END_GET
END_PROPERTY

PROPERTY ProcessExecution : ProcessExecution_e
GET
ProcessExecution := THIS^._ProcessExecution;
END_GET
SET
THIS^._ProcessExecution := ProcessExecution;
END_SET
END_PROPERTY

PROPERTY xBusy : BOOL
GET
xBusy := THIS^.fb_Dose.xOUT_Busy;
END_GET
SET
END_SET
END_PROPERTY

PROPERTY xDone : BOOL
GET
xDone := THIS^.fb_Dose.xOUT_Ready OR THIS^.fb_Dose.xOUT_Done;
END_GET
END_PROPERTY

PROPERTY xMoverPathFree : BOOL
GET
xMoverPathFree := THIS^.fb_Dose.xOUT_MoverFree OR THIS^.fb_Dose.xOUT_Ready OR THIS^.fb_Dose.xOUT_Done;
END_GET
END_PROPERTY

PROPERTY xMoverShouldLeave : BOOL
GET
xMoverShouldLeave := THIS^.fb_Dose.iOUT_Step = ST100_Modify_e.SYNC_MOVER_LEAVE;
END_GET
END_PROPERTY

END_FUNCTION_BLOCK

// ---- POUs/20_AUTO/ST130/FB_ABL_MODIFY_135.TcPOU
FUNCTION_BLOCK FB_ABL_MODIFY_135
(****************************************************************************************)
(*	TITEL				Bezeichnung Ablauf	    										*)
(*	Status				ungetestet                         								*)
(*  Version:			1.0																*)
(*	Beschrieb:			Ablaufbeschreibung												*)
(*																						*)
(*	Steps:																				*)
(*		RESET:=0		Reset der Station												*)
(* 		INIT:=100		Initialisieren													*)
(*		... 			...																*)
(*		READY:=999		Initialisiert, Bereit für Start									*)
(*		START:=1000		Start Zyklisch 													*)
(*		... 			...																*)
(*		DONE:=8000		Letzer Schritt													*)
(*		ERROR:=9000		ALARM/Fehler													*)
(* 	09.09.2019/Dj																		*)
(***********************************Revisionen*******************************************)
(*	dd.mm.yyyy   KZ    x.y			Beschrieb											*)
(****************************************************************************************)

VAR_INPUT
    xIN_Reset       : BOOL;          // Schrittkette zurücksetzen 
    xIN_Init        : BOOL;          // Initialisieren
    xIN_Quit        : BOOL;          // Fehler quittieren 
    xIN_Start       : BOOL;          // Startbefehl
    xIN_Sperre      : BOOL;          // FB Sperren 
    xIN_NextStep    : BOOL;          // Nächsten Schritt ausführen 
    xIN_AlarmAktiv  : BOOL;          // Anlage hat Alarm
    xIN_DryCycle    : BOOL;          // Fahren ohne Teile
    xIN_RestartCYCL : BOOL;          // Zyklus erneut starten im STEP, END, LEERFAHREN
    enIN_State      : enState;       // Status Anlage
    tIN_Timeout     : TIME := T#10s; // Timout

    pxFG_Freigabe : POINTER TO BOOL; //Freigabe von Station

    // Application specific
    iProcessTimeMili1 : UDINT := 5000; // user defined station duration, in milisecond
    iProcessTimeMili2 : UDINT := 5000; // user defined station duration, in milisecond
    Mover            : REFERENCE TO FB_Mover;
    //xIN_MoverInPos  : BOOL;          // Set this flag when a mover is in position and ready to be handled
END_VAR
VAR_OUTPUT
    (* standart Ausgänge *)
    xOUT_ErrFlag     : BOOL;   // Error Flag 
    xOUT_Busy        : BOOL;   // Baustein befindet sich im Ablauf 
    xOUT_Done        : BOOL;   // Baustein hat den Ablauf beendet 		
    xOUT_Ready       : BOOL;   // Ready to begin, should be the same state as done	
    xOUT_Timeout     : BOOL;   // Timeout FB 
    xOUT_InitDone    : BOOL;   // initialisierung fertig
    xOUT_Wait        : BOOL;   // Wartet auf Bedingung
    iOUT_Step        : ST100_Modify_e;    // Aktueller Schritt 
    sOUT_Step        : STRING; // Aktueller Schritt but in string format
    bOUT_Error       : BYTE;   // Fehlernummer

    xOUT_MoverFree   : BOOL;   // The mover is free to move
    //xOUT_MoverNeeded : BOOL;   // A mover is needed by this station to continue its process
    iOUT_ProcessCompletion : INT; //process completion, express in % (0-100)
END_VAR
VAR
    (* Standard *)
    (* Schritt *)
    iLastStep : ST100_Modify_e; // Merker letzter Schritt 
    iPreStep  : ST100_Modify_e; // Schritt zurück nach Alarm 
    iAktStep  : ST100_Modify_e; // aktueller Schritt

    // Trigger Starten 
    rtSTART : R_TRIG;
    // Timer TimeOut 
    TON_Timeout : TON;

    (* Bausteine *)

    (* Spezial *)
    iStartProcessTimeMili : UDINT; // start of the processing time, accurate at 100ns 

END_VAR
VAR CONSTANT
END_VAR

(*******************************************************************)
(* Trigger  *)
(*******************************************************************)
(* Zurücksetzen *)
IF xIN_RESET THEN
    iPreStep  := ST100_Modify_e.RESET;
    iOUT_Step := ST100_Modify_e.RESET;
END_IF;

(* Error Quittieren *)
IF (bOUT_Error <> 0) AND xIN_Quit THEN
    xOUT_ErrFlag := FALSE;
    bOUT_Error   := 0;
    iOUT_Step    := iPreStep;
END_IF;

(*******************************************************************)
(* Timer *)
(*******************************************************************)
TON_Timeout(IN := xIN_NextStep AND (iLastStep = iOUT_Step) (*todo FG *) ,
            PT := tIN_Timeout);

(*******************************************************************)
(* Bausteine *)
(*******************************************************************)

(*******************************************************************)
(* OUTPUTS *)
(*******************************************************************)
// Error Flag 
xOUT_ErrFlag := (bOUT_Error <> 0);
// Baustein befindet sich im Ablauf 
xOUT_Busy := (iOUT_Step > ST100_Modify_e.READY) AND (iOUT_Step < ST100_Modify_e.DONE);
// Baustein hat den Ablauf beendet
xOUT_Done := (iOUT_Step = ST100_Modify_e.DONE);
// Process ready
xOUT_Ready := (iOUT_Step = ST100_Modify_e.READY);
// Timeout FB 				 		
xOUT_Timeout := TON_Timeout.Q;
// Itialisierung fertig			
xOUT_InitDone := (iOUT_Step = ST100_Modify_e.READY);
// Aktueller Schritt			
iOUT_Step := iOUT_Step; //Im Ablauf gesetzt		
sOUT_Step := TO_STRING(iOUT_Step);
//Fehlernummer	 
bOUT_Error := bOUT_Error; //Im Ablauf/FB gesetzt	
(* Warte (alle Schritte wo auf FG oder Teile gewartet wird) *)
xOUT_Wait := (iOUT_Step = ST100_Modify_e.DONE) OR
             (iOUT_Step = ST100_Modify_e.READY) OR
             (iOUT_Step = ST100_Modify_e.START) OR
             (iOUT_Step = ST100_Modify_e.waitOnMover) OR
             (iOUT_Step = ST100_Modify_e.SYNC_MOVER_LEAVE);

xOUT_MoverFree := iOUT_Step = ST100_Modify_e.waitOnMover;

iOUT_ProcessCompletion := F_GetPercent(iAktStep,
                                       ST100_Modify_e.START,
                                       ST100_Modify_e.DONE,
                                       ST100_Modify_e.proceedOperation_1,
                                       ST100_Modify_e.proceedOperation_2,
                                       iStartProcessTimeMili,
                                       TO_DINT(iProcessTimeMili1),
                                       TO_DINT(iProcessTimeMili2));

(*******************************************************************)
(* Ablauf *)
(*******************************************************************)

(* Sperren *)
IF xIN_Sperre THEN
    iPreStep  := ST100_Modify_e.RESET;
    iOUT_Step := ST100_Modify_e.RESET;
    RETURN;
END_IF;

(* Schritt Merker *)
IF iAktStep <> iOUT_Step THEN
    iLastStep := iAktStep;
    iAktStep  := iOUT_Step;
END_IF

(* START *)
rtSTART(CLK := xIN_Start);

(*******************************************************************)
(* Schrittkette  *)
(*******************************************************************)
CASE iOUT_Step OF

(***** RESET *****)
ST100_Modify_e.RESET: (* Schritt 0-99 *)
    //Initialisierungen
    //Start Init Ablauf
    IF xIN_Init THEN
        iOUT_Step := ST100_Modify_e.INIT;
        //Start Manu Ablauf
    ELSIF enIN_State = StateMANU AND xIN_NextStep THEN
        iOUT_Step := ST100_Modify_e.INIT;
    END_IF;

(***** INIT *****)
ST100_Modify_e.INIT: (* Grundstellung ? *)
    IF TRUE THEN
        iOUT_Step := ST100_Modify_e.READY;
    ELSE
        iOUT_Step := ST100_Modify_e.INIT;
    END_IF;

(***** READY / INIT DONE *****)
ST100_Modify_e.READY: (* Start AUTO,END,LEER,STEP *)
    IF xIN_Start THEN //IF rtSTART.Q THEN
        iOUT_Step := ST100_Modify_e.START;
    END_IF

(***** START  ZYKLISCH *****)
ST100_Modify_e.START: (*  *)
    IF xIN_NextStep AND pxFG_Freigabe^ THEN
        iOUT_Step             := ST100_Modify_e.waitOnMover;
        iStartProcessTimeMili := GetTick();
    END_IF;

ST100_Modify_e.waitOnMover: (*  *)
    IF xIN_NextStep AND __ISVALIDREF(Mover) THEN
        iStartProcessTimeMili := GetTick();

        IF Mover.GetLastStationDone() >= INT#135 THEN
            iOUT_Step := ST100_Modify_e.SYNC_MOVER_LEAVE;
        ELSIF Mover.GetLastStationDone() < INT#105 THEN
            iOUT_Step := ST100_Modify_e.SYNC_MOVER_LEAVE;
        ELSE
            IF __ISVALIDREF(Mover) THEN
                IF NOT Mover.SetLastStation(135) THEN
                    ASSERT(0);
                END_IF
            END_IF

            iOUT_Step := ST100_Modify_e.proceedOperation_1;
        END_IF
    END_IF;

ST100_Modify_e.proceedOperation_1: (*  *)
    IF xIN_NextStep AND (GetTick() - iStartProcessTimeMili) >= (iProcessTimeMili1) THEN
        iStartProcessTimeMili := GetTick();
        iOUT_Step             := ST100_Modify_e.proceedOperation_2;
    END_IF

ST100_Modify_e.proceedOperation_2: (*  *)
    IF xIN_NextStep AND (GetTick() - iStartProcessTimeMili) >= (iProcessTimeMili2) THEN
        iOUT_Step := ST100_Modify_e.SYNC_MOVER_LEAVE;
    END_IF;

ST100_Modify_e.SYNC_MOVER_LEAVE:
    // The mover needs to be taken by MoverMan
    IF NOT __ISVALIDREF(Mover) THEN
        iOUT_Step := ST100_Modify_e.DONE;
    END_IF

(***** DONE *****)
ST100_Modify_e.DONE: (* Letzter Schritt  *)
    IF NOT xIN_AlarmAktiv THEN
        //AUTO
        IF (enIN_State = StateAUTO) AND xIN_RestartCYCL THEN
            iOUT_Step := ST100_Modify_e.START;
            //STEP / END / LEERFAHREN restart
        ELSIF (enIN_State < StateAUTO) AND (enIN_State >= enState.StateSTEP) AND xIN_RestartCYCL THEN
            iOUT_Step := ST100_Modify_e.START;
            //STEP / END / LEERFAHREN fertig
        ELSIF (enIN_State = StateREADY) THEN
            iOUT_Step := ST100_Modify_e.READY;
        END_IF;
    END_IF;

(************ ERROR *************)
ST100_Modify_e.ERROR: (* ERROR *) ;

END_CASE;

END_FUNCTION_BLOCK

// ---- POUs/20_AUTO/ST140/FB_AUT_140.TcPOU
FUNCTION_BLOCK FB_AUT_140 EXTENDS FB_AUT_ABSTRACT
(****************************************************************************)
(*	POU_AUT_zxx			Bausteinaufrufe Station	zxx							*)
(*	Status				ungetestet											*)
(*  Version:			1.0													*)
(*	Beschrieb:																*)
(*																			*)
(*	Abläufe:			FB_ABLzxxA		Hauptablauf							*)
(*																			*)
(*																			*)
(* 	25.09.2019/Dj															*)
(****************************************************************************)
(*	dd.mm.yyyy   KZ    x.y			Beschrieb								*)
(****************************************************************************)
VAR_INPUT
    (* spezifische Eingänge *)

END_VAR
VAR_OUTPUT
    (* spezifische Ausgänge *)

END_VAR
VAR
    (* Bausteine *)
    fb_Measure : FB_ABL_140_Measure;

END_VAR

(*******************************************************************)
(* Timer *)
(*******************************************************************)

(*******************************************************************)
(* Flanken / Merker *)
(*******************************************************************)
//MANU CYCLE
IF (enIN_State = StateMANU) AND xIN_ManuCycle THEN
    xManuCycle := TRUE;
END_IF;

IF (enIN_State <> StateMANU) OR xOUT_Done THEN
    xManuCycle := FALSE;
END_IF

//NEXT STEP
xNextStep := (enIN_State > StateSTEP) OR
             ((enIN_State = StateSTEP) AND xIN_Step) OR
             ((enIN_State = StateMANU) AND xManuCycle);

//RESET
xReset := (enIN_State < StateREADY) AND (enIN_State <> StateINIT) AND NOT xManuCycle;

(*******************************************************************)
(* Bausteinaufrufe Abläufe *)
(*******************************************************************)

xRelease := MAIN.MoverMan.IsProcessUsed(THIS^);

fb_Measure(xIN_Reset       := xReset,
           xIN_Init        := xIN_Init,
           xIN_Quit        := xIN_Quit,
           xIN_Start       := enIN_State >= enState.StateLEER AND xRelease,
           xIN_Sperre      := NOT xIN_On,
           xIN_NextStep    := xNextStep,
           xIN_AlarmAktiv  := xIN_AlarmAktiv,
           xIN_DryCycle    := xIN_DryCycle,
           xIN_RestartCYCL := enIN_State >= enState.StateLEER,
           enIN_State      := enIN_State,
           tIN_Timeout     := tIN_Timeout,
           pxFG_Freigabe   := ADR(xRelease),
           Mover           := THIS^.Mover);

(*******************************************************************)
(* Mover reset flags *)
(*******************************************************************)

(*******************************************************************)
(* OUTPUT *)
(*******************************************************************)
xOUT_InitDone := fb_Measure.xOUT_InitDone;
xOUT_Ready    := fb_Measure.xOUT_Ready;
xOUT_Done     := fb_Measure.xOUT_Done;
xOUT_ErrFlag  := fb_Measure.xOUT_ErrFlag;
xOUT_Wait     := fb_Measure.xOUT_Wait;
xOUT_AlarmST  := xOUT_ErrFlag;

(*******************************************************************)
(* Bausteinaufruf Error Station *)
(*******************************************************************)
// POU_ERR_VORLAGE(xIN_QUIT:=xIN_Quit , pstrArIN_ALARM:=ADR(HMI.strArALARM[1]));

(* % of completion of the process *)
PROPERTY iCompletionPC : INT
GET
iCompletionPC := THIS^.fb_Measure.iOUT_ProcessCompletion;
END_GET
END_PROPERTY

PROPERTY ProcessExecution : ProcessExecution_e
GET
ProcessExecution := THIS^._ProcessExecution;
END_GET
SET
THIS^._ProcessExecution := ProcessExecution;
END_SET
END_PROPERTY

PROPERTY xBusy : BOOL
GET
xBusy := THIS^.fb_Measure.xOUT_Busy;
END_GET
SET
END_SET
END_PROPERTY

PROPERTY xDone : BOOL
GET
xDone := THIS^.fb_Measure.xOUT_Ready OR THIS^.fb_Measure.xOUT_Done;
END_GET
END_PROPERTY

PROPERTY xMoverPathFree : BOOL
GET
xMoverPathFree := THIS^.fb_Measure.xOUT_MoverFree OR THIS^.fb_Measure.xOUT_Ready OR THIS^.fb_Measure.xOUT_Done;
END_GET
END_PROPERTY

PROPERTY xMoverShouldLeave : BOOL
GET
xMoverShouldLeave := THIS^.fb_Measure.iOUT_Step = ST140_Measure_e.SYNC_MOVER_LEAVE;
END_GET
END_PROPERTY

END_FUNCTION_BLOCK

// ---- POUs/20_AUTO/ST140/FB_ABL_140_Measure.TcPOU
FUNCTION_BLOCK FB_ABL_140_Measure
(****************************************************************************************)
(*	TITEL				laden kristall- Modul	    										*)
(*	Status				ungetestet                         								*)
(*	Beschrieb:			Ablaufbeschreibung												*)
(*																						*)
(*	Steps:	self-explained using enum													*)
(***********************************Revisionen*******************************************)
(*	see github blames																	*)
(****************************************************************************************)

VAR_INPUT
    xIN_Reset       : BOOL;          // Schrittkette zurücksetzen 
    xIN_Init        : BOOL;          // Initialisieren
    xIN_Quit        : BOOL;          // Fehler quittieren 
    xIN_Start       : BOOL;          // Startbefehl
    xIN_Sperre      : BOOL;          // FB Sperren 
    xIN_NextStep    : BOOL;          // Nächsten Schritt ausführen 
    xIN_AlarmAktiv  : BOOL;          // Anlage hat Alarm
    xIN_DryCycle    : BOOL;          // Fahren ohne Teile
    xIN_RestartCYCL : BOOL;          // Zyklus erneut starten im STEP: END: LEERFAHREN
    enIN_State      : enState;       // Status Anlage
    tIN_Timeout     : TIME := T#10s; // Timout

    pxFG_Freigabe : POINTER TO BOOL; //Freigabe von Station

